LIN {X 0,Y 293.169,Z 768.015,A -85,B 0,C 180,E1 -18492.171,E2 -18492.171} C_VEL
LIN {X 0,Y 292.297,Z 765.8,A -85,B 0,C 180,E1 -18494.106,E2 -18494.106} C_VEL
LIN {X 0,Y 291.883,Z 764.889,A -85,B 0,C 180,E1 -18496.257,E2 -18496.257} C_VEL
LIN {X 0,Y 292.536,Z 764.782,A -85,B 0,C 180,E1 -18498.796,E2 -18498.796} C_VEL
LIN {X 0,Y 294.22,Z 766.186,A -85,B 0,C 180,E1 -18501.347,E2 -18501.347} C_VEL
LIN {X 0,Y 294.782,Z 766.996,A -85,B 0,C 180,E1 -18501.989,E2 -18501.989} C_VEL
LIN {X 0,Y 296.752,Z 771.019,A -85,B 0,C 180,E1 -18504.014,E2 -18504.014} C_VEL
LIN {X 0,Y 298.93,Z 775.634,A -85,B 0,C 180,E1 -18505.733,E2 -18505.733} C_VEL
LIN {X 0,Y 299.613,Z 777.365,A -85,B 0,C 180,E1 -18506.216,E2 -18506.216} C_VEL
LIN {X 0,Y 294.851,Z 808.828,A -85,B 0,C 180,E1 -18507.724,E2 -18507.724} C_VEL
LIN {X 0,Y 292.822,Z 825.485,A -85,B 0,C 180,E1 -18508.733,E2 -18508.733} C_VEL
LIN {X 0,Y 291.112,Z 835.939,A -85,B 0,C 180,E1 -18509.537,E2 -18509.537} C_VEL
LIN {X 0,Y 288.763,Z 847.798,A -85,B 0,C 180,E1 -18510.672,E2 -18510.672} C_VEL
LIN {X 0,Y 285.703,Z 859.648,A -85,B 0,C 180,E1 -18512.136,E2 -18512.136} C_VEL
LIN {X 0,Y 283.074,Z 868.365,A -85,B 0,C 180,E1 -18513.455,E2 -18513.455} C_VEL
LIN {X 0,Y 280.555,Z 875.778,A -85,B 0,C 180,E1 -18514.795,E2 -18514.795} C_VEL
LIN {X 0,Y 277.606,Z 883.425,A -85,B 0,C 180,E1 -18516.468,E2 -18516.468} C_VEL
LIN {X 0,Y 275.249,Z 888.923,A -85,B 0,C 180,E1 -18517.876,E2 -18517.876} C_VEL
LIN {X 0,Y 272.596,Z 894.53,A -85,B 0,C 180,E1 -18519.632,E2 -18519.632} C_VEL
LIN {X 0,Y 269.635,Z 899.978,A -85,B 0,C 180,E1 -18521.773,E2 -18521.773} C_VEL
LIN {X 0,Y 266.922,Z 904.27,A -85,B 0,C 180,E1 -18523.951,E2 -18523.951} C_VEL
LIN {X 0,Y 264.533,Z 907.404,A -85,B 0,C 180,E1 -18526.166,E2 -18526.166} C_VEL
LIN {X 0,Y 263.113,Z 908.967,A -85,B 0,C 180,E1 -18527.661,E2 -18527.661} C_VEL
LIN {X 0,Y 261.774,Z 910.083,A -85,B 0,C 180,E1 -18529.168,E2 -18529.168} C_VEL
LIN {X 0,Y 259.678,Z 910.938,A -85,B 0,C 180,E1 -18532.223,E2 -18532.223} C_VEL
LIN {X 0,Y 258.847,Z 910.711,A -85,B 0,C 180,E1 -18533.765,E2 -18533.765} C_VEL
LIN {X 0,Y 258.245,Z 910.062,A -85,B 0,C 180,E1 -18535.317,E2 -18535.317} C_VEL
LIN {X 0,Y 257.539,Z 908.966,A -85,B 0,C 180,E1 -18536.871,E2 -18536.871} C_VEL
LIN {X 0,Y 257.125,Z 907.432,A -85,B 0,C 180,E1 -18538.434,E2 -18538.434} C_VEL
LIN {X 0,Y 256.51,Z 904.341,A -85,B 0,C 180,E1 -18540.785,E2 -18540.785} C_VEL
LIN {X 0,Y 256.12,Z 900.192,A -85,B 0,C 180,E1 -18543.146,E2 -18543.146} C_VEL
LIN {X 0,Y 256.313,Z 893.788,A -85,B 0,C 180,E1 -18545.902,E2 -18545.902} C_VEL
LIN {X 0,Y 256.713,Z 886.811,A -85,B 0,C 180,E1 -18548.264,E2 -18548.264} C_VEL
LIN {X 0,Y 257.046,Z 880.2,A -85,B 0,C 180,E1 -18550.133,E2 -18550.133} C_VEL
LIN {X 0,Y 257.479,Z 873.243,A -85,B 0,C 180,E1 -18551.813,E2 -18551.813} C_VEL
LIN {X 0,Y 258.123,Z 864.599,A -85,B 0,C 180,E1 -18553.582,E2 -18553.582} C_VEL
LIN {X 0,Y 258.704,Z 855.499,A -85,B 0,C 180,E1 -18555.158,E2 -18555.158} C_VEL
LIN {X 0,Y 259.349,Z 846.095,A -85,B 0,C 180,E1 -18556.531,E2 -18556.531} C_VEL
LIN {X 0,Y 259.959,Z 836.514,A -85,B 0,C 180,E1 -18557.707,E2 -18557.707} C_VEL
LIN {X 0,Y 260.523,Z 826.952,A -85,B 0,C 180,E1 -18558.684,E2 -18558.684} C_VEL
LIN {X 0,Y 260.988,Z 815.785,A -85,B 0,C 180,E1 -18559.601,E2 -18559.601} C_VEL
LIN {X 0,Y 261.302,Z 804.987,A -85,B 0,C 180,E1 -18560.287,E2 -18560.287} C_VEL
LIN {X 0,Y 261.675,Z 788.222,A -85,B 0,C 180,E1 -18561.053,E2 -18561.053} C_VEL
LIN {X 0,Y 262.992,Z 743.404,A -85,B 0,C 180,E1 -18562.898,E2 -18562.898} C_VEL
LIN {X 0,Y 256.201,Z 720.571,A -85,B 0,C 180,E1 -18564.225,E2 -18564.225} C_VEL
LIN {X 0,Y 256.107,Z 720.581,A -85,B 0,C 180,E1 -18568.568,E2 -18568.568} C_VEL
LIN {X 0,Y 256.095,Z 720.583,A -85,B 0,C 180,E1 -18571.695,E2 -18571.695} C_VEL
LIN {X 0,Y 256.104,Z 720.582,A -85,B 0,C 180,E1 -18575.19,E2 -18575.19} C_VEL
LIN {X 0,Y 256.089,Z 720.581,A -85,B 0,C 180,E1 -18579.139,E2 -18579.139} C_VEL
LIN {X 0,Y 256.046,Z 720.585,A -85,B 0,C 180,E1 -18583.331,E2 -18583.331} C_VEL
LIN {X 0,Y 256.056,Z 720.583,A -85,B 0,C 180,E1 -18587.823,E2 -18587.823} C_VEL
LIN {X 0,Y 256.086,Z 720.578,A -85,B 0,C 180,E1 -18590.85,E2 -18590.85} C_VEL
LIN {X 0,Y 256.1,Z 720.577,A -85,B 0,C 180,E1 -18594.8,E2 -18594.8} C_VEL
LIN {X 0,Y 256.118,Z 720.772,A -85,B 0,C 180,E1 -18598.348,E2 -18598.348} C_VEL
LIN {X 0,Y 257.16,Z 723.493,A -85,B 0,C 180,E1 -18598.585,E2 -18598.585} C_VEL
LIN {X 0,Y 258.744,Z 726.144,A -85,B 0,C 180,E1 -18598.893,E2 -18598.893} C_VEL
LIN {X 0,Y 266.211,Z 739.942,A -85,B 0,C 180,E1 -18600.322,E2 -18600.322} C_VEL
LIN {X 0,Y 273.123,Z 754.427,A -85,B 0,C 180,E1 -18601.608,E2 -18601.608} C_VEL
LIN {X 0,Y 273.856,Z 756.115,A -85,B 0,C 180,E1 -18601.745,E2 -18601.745} C_VEL
LIN {X 0,Y 272.925,Z 794.728,A -85,B 0,C 180,E1 -18602.771,E2 -18602.771} C_VEL
LIN {X 0,Y 272.718,Z 809.458,A -85,B 0,C 180,E1 -18603.281,E2 -18603.281} C_VEL
LIN {X 0,Y 272.187,Z 821.386,A -85,B 0,C 180,E1 -18603.954,E2 -18603.954} C_VEL
LIN {X 0,Y 271.062,Z 834.416,A -85,B 0,C 180,E1 -18605.002,E2 -18605.002} C_VEL
LIN {X 0,Y 269.714,Z 845.924,A -85,B 0,C 180,E1 -18606.238,E2 -18606.238} C_VEL
LIN {X 0,Y 268.04,Z 856.353,A -85,B 0,C 180,E1 -18607.645,E2 -18607.645} C_VEL
LIN {X 0,Y 266.537,Z 865.181,A -85,B 0,C 180,E1 -18609.138,E2 -18609.138} C_VEL
LIN {X 0,Y 264.837,Z 874.215,A -85,B 0,C 180,E1 -18611.02,E2 -18611.02} C_VEL
LIN {X 0,Y 262.82,Z 882.996,A -85,B 0,C 180,E1 -18613.284,E2 -18613.284} C_VEL
LIN {X 0,Y 260.98,Z 890.664,A -85,B 0,C 180,E1 -18615.803,E2 -18615.803} C_VEL
LIN {X 0,Y 259.741,Z 896.427,A -85,B 0,C 180,E1 -18618.282,E2 -18618.282} C_VEL
LIN {X 0,Y 259.045,Z 899.362,A -85,B 0,C 180,E1 -18619.833,E2 -18619.833} C_VEL
LIN {X 0,Y 257.846,Z 902.921,A -85,B 0,C 180,E1 -18622.157,E2 -18622.157} C_VEL
LIN {X 0,Y 257.338,Z 904.743,A -85,B 0,C 180,E1 -18623.718,E2 -18623.718} C_VEL
LIN {X 0,Y 256.95,Z 907.051,A -85,B 0,C 180,E1 -18626.854,E2 -18626.854} C_VEL
LIN {X 0,Y 256.667,Z 907.89,A -85,B 0,C 180,E1 -18629.99,E2 -18629.99} C_VEL
LIN {X 0,Y 256.946,Z 907.124,A -85,B 0,C 180,E1 -18633.125,E2 -18633.125} C_VEL
LIN {X 0,Y 257.317,Z 904.893,A -85,B 0,C 180,E1 -18636.261,E2 -18636.261} C_VEL
LIN {X 0,Y 258.168,Z 902.073,A -85,B 0,C 180,E1 -18638.6,E2 -18638.6} C_VEL
LIN {X 0,Y 259.312,Z 898.243,A -85,B 0,C 180,E1 -18640.925,E2 -18640.925} C_VEL
LIN {X 0,Y 260.559,Z 892.768,A -85,B 0,C 180,E1 -18643.489,E2 -18643.489} C_VEL
LIN {X 0,Y 262.202,Z 885.953,A -85,B 0,C 180,E1 -18645.935,E2 -18645.935} C_VEL
LIN {X 0,Y 264.102,Z 877.921,A -85,B 0,C 180,E1 -18648.209,E2 -18648.209} C_VEL
LIN {X 0,Y 265.782,Z 869.698,A -85,B 0,C 180,E1 -18650.094,E2 -18650.094} C_VEL
LIN {X 0,Y 267.597,Z 859.522,A -85,B 0,C 180,E1 -18651.966,E2 -18651.966} C_VEL
LIN {X 0,Y 269.347,Z 849.047,A -85,B 0,C 180,E1 -18653.488,E2 -18653.488} C_VEL
LIN {X 0,Y 270.844,Z 837.769,A -85,B 0,C 180,E1 -18654.788,E2 -18654.788} C_VEL
LIN {X 0,Y 272.079,Z 825.822,A -85,B 0,C 180,E1 -18655.829,E2 -18655.829} C_VEL
LIN {X 0,Y 272.637,Z 813.644,A -85,B 0,C 180,E1 -18656.629,E2 -18656.629} C_VEL
LIN {X 0,Y 272.938,Z 800.891,A -85,B 0,C 180,E1 -18657.169,E2 -18657.169} C_VEL
LIN {X 0,Y 273.85,Z 760.256,A -85,B 0,C 180,E1 -18658.263,E2 -18658.263} C_VEL
LIN {X 0,Y 273.819,Z 755.874,A -85,B 0,C 180,E1 -18658.396,E2 -18658.396} C_VEL
LIN {X 0,Y 266.835,Z 741.021,A -85,B 0,C 180,E1 -18659.697,E2 -18659.697} C_VEL
LIN {X 0,Y 259.331,Z 727.24,A -85,B 0,C 180,E1 -18661.126,E2 -18661.126} C_VEL
LIN {X 0,Y 256.33,Z 721.817,A -85,B 0,C 180,E1 -18661.725,E2 -18661.725} C_VEL
LIN {X 0,Y 256.065,Z 720.589,A -85,B 0,C 180,E1 -18661.825,E2 -18661.825} C_VEL
LIN {X 0,Y 256.09,Z 720.585,A -85,B 0,C 180,E1 -18665.176,E2 -18665.176} C_VEL
LIN {X 0,Y 256.074,Z 720.569,A -85,B 0,C 180,E1 -18669.125,E2 -18669.125} C_VEL
LIN {X 0,Y 256.102,Z 720.573,A -85,B 0,C 180,E1 -18673.301,E2 -18673.301} C_VEL
LIN {X 0,Y 256.117,Z 720.579,A -85,B 0,C 180,E1 -18677.788,E2 -18677.788} C_VEL
LIN {X 0,Y 256.063,Z 720.583,A -85,B 0,C 180,E1 -18680.856,E2 -18680.856} C_VEL
LIN {X 0,Y 256.071,Z 720.583,A -85,B 0,C 180,E1 -18684.805,E2 -18684.805} C_VEL
LIN {X 0,Y 256.04,Z 720.59,A -85,B 0,C 180,E1 -18688.565,E2 -18688.565} C_VEL
LIN {X 0,Y 256.083,Z 720.578,A -85,B 0,C 180,E1 -18692.189,E2 -18692.189} C_VEL
LIN {X 0,Y 256.085,Z 720.576,A -85,B 0,C 180,E1 -18695.691,E2 -18695.691} C_VEL
LIN {X 0,Y 256.105,Z 720.583,A -85,B 0,C 180,E1 -18699.099,E2 -18699.099} C_VEL
LIN {X 0,Y 256.218,Z 720.56,A -85,B 0,C 180,E1 -18704.08,E2 -18704.08} C_VEL
LIN {X 0,Y 256.246,Z 720.551,A -85,B 0,C 180,E1 -18708.931,E2 -18708.931} C_VEL
LIN {X 0,Y 256.33,Z 720.542,A -85,B 0,C 180,E1 -18710.1,E2 -18710.1} C_VEL
LIN {X 0,Y 255.761,Z 720.627,A -85,B 0,C 180,E1 -18711.411,E2 -18711.411} C_VEL
LIN {X 0,Y 252.905,Z 720.983,A -85,B 0,C 180,E1 -18713.546,E2 -18713.546} C_VEL
LIN {X 0,Y 250.46,Z 721.279,A -85,B 0,C 180,E1 -18715.286,E2 -18715.286} C_VEL
LIN {X 0,Y 249.472,Z 721.398,A -85,B 0,C 180,E1 -18716.636,E2 -18716.636} C_VEL
LIN {X 0,Y 249.428,Z 721.404,A -85,B 0,C 180,E1 -18717.093,E2 -18717.093} C_VEL
LIN {X 0,Y 249.67,Z 721.389,A -85,B 0,C 180,E1 -18720,E2 -18720} C_VEL
LIN {X 0,Y 249.401,Z 721.408,A -85,B 0,C 180,E1 -18723.231,E2 -18723.231} C_VEL
LIN {X 0,Y 249.406,Z 721.412,A -85,B 0,C 180,E1 -18728.1,E2 -18728.1} C_VEL
LIN {X 0,Y 249.189,Z 721.445,A -85,B 0,C 180,E1 -18731.386,E2 -18731.386} C_VEL
LIN {X 0,Y 249.158,Z 721.445,A -85,B 0,C 180,E1 -18736.507,E2 -18736.507} C_VEL
LIN {X 0,Y 249.028,Z 721.452,A -85,B 0,C 180,E1 -18741.524,E2 -18741.524} C_VEL
LIN {X 0,Y 249.073,Z 721.448,A -85,B 0,C 180,E1 -18745.487,E2 -18745.487} C_VEL
LIN {X 0,Y 249.019,Z 721.464,A -85,B 0,C 180,E1 -18748.996,E2 -18748.996} C_VEL
LIN {X 0,Y 248.984,Z 721.47,A -85,B 0,C 180,E1 -18752.433,E2 -18752.433} C_VEL
LIN {X 0,Y 249.025,Z 721.464,A -85,B 0,C 180,E1 -18756.346,E2 -18756.346} C_VEL
LIN {X 0,Y 249.039,Z 721.452,A -85,B 0,C 180,E1 -18760.472,E2 -18760.472} C_VEL
LIN {X 0,Y 249.032,Z 721.47,A -85,B 0,C 180,E1 -18764.321,E2 -18764.321} C_VEL
LIN {X 0,Y 252.137,Z 732.401,A -85,B 0,C 180,E1 -18768.349,E2 -18768.349} C_VEL
LIN {X 0,Y 254.654,Z 742.514,A -85,B 0,C 180,E1 -18771.768,E2 -18771.768} C_VEL
LIN {X 0,Y 256.98,Z 753.129,A -85,B 0,C 180,E1 -18775.13,E2 -18775.13} C_VEL
LIN {X 0,Y 257.957,Z 759.353,A -85,B 0,C 180,E1 -18776.997,E2 -18776.997} C_VEL
LIN {X 0,Y 257.44,Z 762.214,A -85,B 0,C 180,E1 -18777.75,E2 -18777.75} C_VEL
LIN {X 0,Y 261.25,Z 791.203,A -85,B 0,C 180,E1 -18779.183,E2 -18779.183} C_VEL
LIN {X 0,Y 264.207,Z 821.563,A -85,B 0,C 180,E1 -18780.474,E2 -18780.474} C_VEL
LIN {X 0,Y 265.313,Z 838.589,A -85,B 0,C 180,E1 -18781.116,E2 -18781.116} C_VEL
LIN {X 0,Y 264.068,Z 874.188,A -85,B 0,C 180,E1 -18782.092,E2 -18782.092} C_VEL
LIN {X 0,Y 262.845,Z 887.976,A -85,B 0,C 180,E1 -18782.755,E2 -18782.755} C_VEL
LIN {X 0,Y 261.319,Z 900.557,A -85,B 0,C 180,E1 -18783.67,E2 -18783.67} C_VEL
LIN {X 0,Y 259.44,Z 911.71,A -85,B 0,C 180,E1 -18784.758,E2 -18784.758} C_VEL
LIN {X 0,Y 257.126,Z 923.35,A -85,B 0,C 180,E1 -18786.237,E2 -18786.237} C_VEL
LIN {X 0,Y 254.911,Z 933.879,A -85,B 0,C 180,E1 -18787.949,E2 -18787.949} C_VEL
LIN {X 0,Y 252.942,Z 942.516,A -85,B 0,C 180,E1 -18789.69,E2 -18789.69} C_VEL
LIN {X 0,Y 251.298,Z 950.546,A -85,B 0,C 180,E1 -18791.674,E2 -18791.674} C_VEL
LIN {X 0,Y 249.89,Z 957.229,A -85,B 0,C 180,E1 -18793.678,E2 -18793.678} C_VEL
LIN {X 0,Y 248.763,Z 963.864,A -85,B 0,C 180,E1 -18796.117,E2 -18796.117} C_VEL
LIN {X 0,Y 248.083,Z 969.178,A -85,B 0,C 180,E1 -18798.574,E2 -18798.574} C_VEL
LIN {X 0,Y 247.895,Z 973.364,A -85,B 0,C 180,E1 -18801.041,E2 -18801.041} C_VEL
LIN {X 0,Y 248.045,Z 976.5,A -85,B 0,C 180,E1 -18803.504,E2 -18803.504} C_VEL
LIN {X 0,Y 248.285,Z 978.015,A -85,B 0,C 180,E1 -18805.14,E2 -18805.14} C_VEL
LIN {X 0,Y 248.498,Z 979.1,A -85,B 0,C 180,E1 -18806.768,E2 -18806.768} C_VEL
LIN {X 0,Y 248.69,Z 979.769,A -85,B 0,C 180,E1 -18808.391,E2 -18808.391} C_VEL
LIN {X 0,Y 248.88,Z 980.017,A -85,B 0,C 180,E1 -18810.011,E2 -18810.011} C_VEL
LIN {X 0,Y 248.689,Z 979.752,A -85,B 0,C 180,E1 -18811.63,E2 -18811.63} C_VEL
LIN {X 0,Y 248.494,Z 979.072,A -85,B 0,C 180,E1 -18813.253,E2 -18813.253} C_VEL
LIN {X 0,Y 248.273,Z 977.974,A -85,B 0,C 180,E1 -18814.882,E2 -18814.882} C_VEL
LIN {X 0,Y 247.98,Z 975.552,A -85,B 0,C 180,E1 -18817.281,E2 -18817.281} C_VEL
LIN {X 0,Y 248.209,Z 969.865,A -85,B 0,C 180,E1 -18822.271,E2 -18822.271} C_VEL
LIN {X 0,Y 249.089,Z 966.281,A -85,B 0,C 180,E1 -18824.72,E2 -18824.72} C_VEL
LIN {X 0,Y 250.863,Z 960.397,A -85,B 0,C 180,E1 -18827.727,E2 -18827.727} C_VEL
LIN {X 0,Y 253.032,Z 955.019,A -85,B 0,C 180,E1 -18829.902,E2 -18829.902} C_VEL
LIN {X 0,Y 255.726,Z 948.036,A -85,B 0,C 180,E1 -18832.212,E2 -18832.212} C_VEL
LIN {X 0,Y 258.534,Z 941.236,A -85,B 0,C 180,E1 -18834.074,E2 -18834.074} C_VEL
LIN {X 0,Y 262.541,Z 931.503,A -85,B 0,C 180,E1 -18836.221,E2 -18836.221} C_VEL
LIN {X 0,Y 265.938,Z 922.997,A -85,B 0,C 180,E1 -18837.77,E2 -18837.77} C_VEL
LIN {X 0,Y 269.691,Z 912.988,A -85,B 0,C 180,E1 -18839.259,E2 -18839.259} C_VEL
LIN {X 0,Y 273.427,Z 902.615,A -85,B 0,C 180,E1 -18840.516,E2 -18840.516} C_VEL
LIN {X 0,Y 276.85,Z 891.854,A -85,B 0,C 180,E1 -18841.581,E2 -18841.581} C_VEL
LIN {X 0,Y 279.987,Z 880.8,A -85,B 0,C 180,E1 -18842.457,E2 -18842.457} C_VEL
LIN {X 0,Y 283.535,Z 866.175,A -85,B 0,C 180,E1 -18843.373,E2 -18843.373} C_VEL
LIN {X 0,Y 287.026,Z 844.8,A -85,B 0,C 180,E1 -18844.388,E2 -18844.388} C_VEL
LIN {X 0,Y 289.011,Z 825.027,A -85,B 0,C 180,E1 -18845.714,E2 -18845.714} C_VEL
LIN {X 0,Y 290.09,Z 809.979,A -85,B 0,C 180,E1 -18847.027,E2 -18847.027} C_VEL
LIN {X 0,Y 291.339,Z 791.88,A -85,B 0,C 180,E1 -18848.883,E2 -18848.883} C_VEL
LIN {X 0,Y 291.656,Z 785.798,A -85,B 0,C 180,E1 -18849.649,E2 -18849.649} C_VEL
LIN {X 0,Y 291.112,Z 776.146,A -85,B 0,C 180,E1 -18852.13,E2 -18852.13} C_VEL
LIN {X 0,Y 291.05,Z 774.422,A -85,B 0,C 180,E1 -18852.673,E2 -18852.673} C_VEL
LIN {X 0,Y 290.487,Z 772.629,A -85,B 0,C 180,E1 -18854.213,E2 -18854.213} C_VEL
LIN {X 0,Y 290.166,Z 771.711,A -85,B 0,C 180,E1 -18856.613,E2 -18856.613} C_VEL
LIN {X 0,Y 290.991,Z 771.836,A -85,B 0,C 180,E1 -18859.3,E2 -18859.3} C_VEL
LIN {X 0,Y 292.489,Z 773.149,A -85,B 0,C 180,E1 -18861.409,E2 -18861.409} C_VEL
LIN {X 0,Y 294.44,Z 777.474,A -85,B 0,C 180,E1 -18863.641,E2 -18863.641} C_VEL
LIN {X 0,Y 296.109,Z 781.305,A -85,B 0,C 180,E1 -18865.099,E2 -18865.099} C_VEL
LIN {X 0,Y 291.176,Z 812.172,A -85,B 0,C 180,E1 -18866.642,E2 -18866.642} C_VEL
LIN {X 0,Y 288.986,Z 828.026,A -85,B 0,C 180,E1 -18867.654,E2 -18867.654} C_VEL
LIN {X 0,Y 286.813,Z 840.119,A -85,B 0,C 180,E1 -18868.62,E2 -18868.62} C_VEL
LIN {X 0,Y 283.873,Z 852.515,A -85,B 0,C 180,E1 -18869.911,E2 -18869.911} C_VEL
LIN {X 0,Y 281.006,Z 862.498,A -85,B 0,C 180,E1 -18871.22,E2 -18871.22} C_VEL
LIN {X 0,Y 278.195,Z 870.951,A -85,B 0,C 180,E1 -18872.545,E2 -18872.545} C_VEL
LIN {X 0,Y 275.496,Z 878.087,A -85,B 0,C 180,E1 -18873.893,E2 -18873.893} C_VEL
LIN {X 0,Y 273.201,Z 883.79,A -85,B 0,C 180,E1 -18875.14,E2 -18875.14} C_VEL
LIN {X 0,Y 270.45,Z 889.739,A -85,B 0,C 180,E1 -18876.653,E2 -18876.653} C_VEL
LIN {X 0,Y 267.54,Z 895.423,A -85,B 0,C 180,E1 -18878.422,E2 -18878.422} C_VEL
LIN {X 0,Y 264.326,Z 900.969,A -85,B 0,C 180,E1 -18880.588,E2 -18880.588} C_VEL
LIN {X 0,Y 261.376,Z 905.28,A -85,B 0,C 180,E1 -18882.796,E2 -18882.796} C_VEL
LIN {X 0,Y 259.59,Z 907.646,A -85,B 0,C 180,E1 -18884.292,E2 -18884.292} C_VEL
LIN {X 0,Y 257.943,Z 909.391,A -85,B 0,C 180,E1 -18885.805,E2 -18885.805} C_VEL
LIN {X 0,Y 255.022,Z 911.73,A -85,B 0,C 180,E1 -18888.877,E2 -18888.877} C_VEL
LIN {X 0,Y 252.781,Z 912.262,A -85,B 0,C 180,E1 -18892.009,E2 -18892.009} C_VEL
LIN {X 0,Y 251.897,Z 911.904,A -85,B 0,C 180,E1 -18893.592,E2 -18893.592} C_VEL
LIN {X 0,Y 251.266,Z 911.066,A -85,B 0,C 180,E1 -18895.187,E2 -18895.187} C_VEL
LIN {X 0,Y 250.07,Z 908.213,A -85,B 0,C 180,E1 -18898.39,E2 -18898.39} C_VEL
LIN {X 0,Y 249.444,Z 904.875,A -85,B 0,C 180,E1 -18900.807,E2 -18900.807} C_VEL
LIN {X 0,Y 249.05,Z 900.432,A -85,B 0,C 180,E1 -18903.236,E2 -18903.236} C_VEL
LIN {X 0,Y 249.168,Z 894.774,A -85,B 0,C 180,E1 -18905.666,E2 -18905.666} C_VEL
LIN {X 0,Y 249.547,Z 888.382,A -85,B 0,C 180,E1 -18907.907,E2 -18907.907} C_VEL
LIN {X 0,Y 249.854,Z 882.301,A -85,B 0,C 180,E1 -18909.716,E2 -18909.716} C_VEL
LIN {X 0,Y 250.361,Z 874.143,A -85,B 0,C 180,E1 -18911.743,E2 -18911.743} C_VEL
LIN {X 0,Y 251.016,Z 865.436,A -85,B 0,C 180,E1 -18913.561,E2 -18913.561} C_VEL
LIN {X 0,Y 251.632,Z 856.273,A -85,B 0,C 180,E1 -18915.179,E2 -18915.179} C_VEL
LIN {X 0,Y 252.255,Z 846.781,A -85,B 0,C 180,E1 -18916.593,E2 -18916.593} C_VEL
LIN {X 0,Y 252.875,Z 837.104,A -85,B 0,C 180,E1 -18917.801,E2 -18917.801} C_VEL
LIN {X 0,Y 253.496,Z 826.357,A -85,B 0,C 180,E1 -18918.907,E2 -18918.907} C_VEL
LIN {X 0,Y 253.981,Z 814.935,A -85,B 0,C 180,E1 -18919.845,E2 -18919.845} C_VEL
LIN {X 0,Y 254.342,Z 801.66,A -85,B 0,C 180,E1 -18920.667,E2 -18920.667} C_VEL
LIN {X 0,Y 255.9,Z 750.146,A -85,B 0,C 180,E1 -18922.906,E2 -18922.906} C_VEL
LIN {X 0,Y 255.927,Z 744.55,A -85,B 0,C 180,E1 -18923.151,E2 -18923.151} C_VEL
LIN {X 0,Y 249.155,Z 721.448,A -85,B 0,C 180,E1 -18924.511,E2 -18924.511} C_VEL
LIN {X 0,Y 249.054,Z 721.463,A -85,B 0,C 180,E1 -18928.966,E2 -18928.966} C_VEL
LIN {X 0,Y 249.052,Z 721.462,A -85,B 0,C 180,E1 -18932.423,E2 -18932.423} C_VEL
LIN {X 0,Y 249.037,Z 721.46,A -85,B 0,C 180,E1 -18936.345,E2 -18936.345} C_VEL
LIN {X 0,Y 249.004,Z 721.465,A -85,B 0,C 180,E1 -18940.479,E2 -18940.479} C_VEL
LIN {X 0,Y 248.986,Z 721.464,A -85,B 0,C 180,E1 -18944.884,E2 -18944.884} C_VEL
LIN {X 0,Y 249.002,Z 721.463,A -85,B 0,C 180,E1 -18947.349,E2 -18947.349} C_VEL
LIN {X 0,Y 249.066,Z 721.453,A -85,B 0,C 180,E1 -18952.194,E2 -18952.194} C_VEL
LIN {X 0,Y 249.06,Z 721.454,A -85,B 0,C 180,E1 -18956.606,E2 -18956.606} C_VEL
LIN {X 0,Y 249.029,Z 721.457,A -85,B 0,C 180,E1 -18957.292,E2 -18957.292} C_VEL
LIN {X 0,Y 250.041,Z 724.295,A -85,B 0,C 180,E1 -18957.569,E2 -18957.569} C_VEL
LIN {X 0,Y 251.872,Z 727.362,A -85,B 0,C 180,E1 -18957.946,E2 -18957.946} C_VEL
LIN {X 0,Y 258.693,Z 739.507,A -85,B 0,C 180,E1 -18959.314,E2 -18959.314} C_VEL
LIN {X 0,Y 266.732,Z 756.106,A -85,B 0,C 180,E1 -18960.882,E2 -18960.882} C_VEL
LIN {X 0,Y 267.626,Z 758.075,A -85,B 0,C 180,E1 -18961.053,E2 -18961.053} C_VEL
LIN {X 0,Y 266.696,Z 795.311,A -85,B 0,C 180,E1 -18962.067,E2 -18962.067} C_VEL
LIN {X 0,Y 266.436,Z 810.923,A -85,B 0,C 180,E1 -18962.62,E2 -18962.62} C_VEL
LIN {X 0,Y 265.806,Z 823.711,A -85,B 0,C 180,E1 -18963.386,E2 -18963.386} C_VEL
LIN {X 0,Y 264.592,Z 836.502,A -85,B 0,C 180,E1 -18964.462,E2 -18964.462} C_VEL
LIN {X 0,Y 263.111,Z 848.07,A -85,B 0,C 180,E1 -18965.757,E2 -18965.757} C_VEL
LIN {X 0,Y 261.392,Z 858.529,A -85,B 0,C 180,E1 -18967.254,E2 -18967.254} C_VEL
LIN {X 0,Y 259.577,Z 868.12,A -85,B 0,C 180,E1 -18968.968,E2 -18968.968} C_VEL
LIN {X 0,Y 257.855,Z 876.811,A -85,B 0,C 180,E1 -18970.9,E2 -18970.9} C_VEL
LIN {X 0,Y 255.798,Z 885.31,A -85,B 0,C 180,E1 -18973.223,E2 -18973.223} C_VEL
LIN {X 0,Y 254.041,Z 892.069,A -85,B 0,C 180,E1 -18975.573,E2 -18975.573} C_VEL
LIN {X 0,Y 252.863,Z 897.431,A -85,B 0,C 180,E1 -18977.958,E2 -18977.958} C_VEL
LIN {X 0,Y 252.131,Z 900.366,A -85,B 0,C 180,E1 -18979.551,E2 -18979.551} C_VEL
LIN {X 0,Y 250.886,Z 903.924,A -85,B 0,C 180,E1 -18981.938,E2 -18981.938} C_VEL
LIN {X 0,Y 250.353,Z 905.746,A -85,B 0,C 180,E1 -18983.542,E2 -18983.542} C_VEL
LIN {X 0,Y 249.934,Z 908.054,A -85,B 0,C 180,E1 -18986.766,E2 -18986.766} C_VEL
LIN {X 0,Y 249.639,Z 908.893,A -85,B 0,C 180,E1 -18989.989,E2 -18989.989} C_VEL
LIN {X 0,Y 249.929,Z 908.126,A -85,B 0,C 180,E1 -18993.213,E2 -18993.213} C_VEL
LIN {X 0,Y 250.331,Z 905.895,A -85,B 0,C 180,E1 -18996.437,E2 -18996.437} C_VEL
LIN {X 0,Y 251.222,Z 903.074,A -85,B 0,C 180,E1 -18998.84,E2 -18998.84} C_VEL
LIN {X 0,Y 252.415,Z 899.245,A -85,B 0,C 180,E1 -19001.227,E2 -19001.227} C_VEL
LIN {X 0,Y 253.73,Z 893.769,A -85,B 0,C 180,E1 -19003.859,E2 -19003.859} C_VEL
LIN {X 0,Y 255.451,Z 886.953,A -85,B 0,C 180,E1 -19006.367,E2 -19006.367} C_VEL
LIN {X 0,Y 257.435,Z 878.921,A -85,B 0,C 180,E1 -19008.698,E2 -19008.698} C_VEL
LIN {X 0,Y 259.193,Z 870.698,A -85,B 0,C 180,E1 -19010.627,E2 -19010.627} C_VEL
LIN {X 0,Y 261.092,Z 860.521,A -85,B 0,C 180,E1 -19012.543,E2 -19012.543} C_VEL
LIN {X 0,Y 262.916,Z 850.044,A -85,B 0,C 180,E1 -19014.099,E2 -19014.099} C_VEL
LIN {X 0,Y 264.481,Z 838.765,A -85,B 0,C 180,E1 -19015.427,E2 -19015.427} C_VEL
LIN {X 0,Y 265.77,Z 826.816,A -85,B 0,C 180,E1 -19016.489,E2 -19016.489} C_VEL
LIN {X 0,Y 266.379,Z 814.229,A -85,B 0,C 180,E1 -19017.33,E2 -19017.33} C_VEL
LIN {X 0,Y 266.701,Z 801.485,A -85,B 0,C 180,E1 -19017.873,E2 -19017.873} C_VEL
LIN {X 0,Y 267.6,Z 761.77,A -85,B 0,C 180,E1 -19018.969,E2 -19018.969} C_VEL
LIN {X 0,Y 267.635,Z 758.009,A -85,B 0,C 180,E1 -19019.079,E2 -19019.079} C_VEL
LIN {X 0,Y 260.781,Z 743.445,A -85,B 0,C 180,E1 -19020.413,E2 -19020.413} C_VEL
LIN {X 0,Y 252.565,Z 728.492,A -85,B 0,C 180,E1 -19022.053,E2 -19022.053} C_VEL
LIN {X 0,Y 249.317,Z 722.816,A -85,B 0,C 180,E1 -19022.732,E2 -19022.732} C_VEL
LIN {X 0,Y 249.023,Z 721.466,A -85,B 0,C 180,E1 -19022.843,E2 -19022.843} C_VEL
LIN {X 0,Y 249.042,Z 721.462,A -85,B 0,C 180,E1 -19026.327,E2 -19026.327} C_VEL
LIN {X 0,Y 249.047,Z 721.461,A -85,B 0,C 180,E1 -19030.452,E2 -19030.452} C_VEL
LIN {X 0,Y 249.055,Z 721.457,A -85,B 0,C 180,E1 -19032.803,E2 -19032.803} C_VEL
LIN {X 0,Y 249.055,Z 721.455,A -85,B 0,C 180,E1 -19037.371,E2 -19037.371} C_VEL
LIN {X 0,Y 249.006,Z 721.461,A -85,B 0,C 180,E1 -19041.615,E2 -19041.615} C_VEL
LIN {X 0,Y 249.011,Z 721.457,A -85,B 0,C 180,E1 -19045.634,E2 -19045.634} C_VEL
LIN {X 0,Y 248.995,Z 721.466,A -85,B 0,C 180,E1 -19049.465,E2 -19049.465} C_VEL
LIN {X 0,Y 249.013,Z 721.465,A -85,B 0,C 180,E1 -19053.155,E2 -19053.155} C_VEL
LIN {X 0,Y 249.004,Z 721.455,A -85,B 0,C 180,E1 -19056.725,E2 -19056.725} C_VEL
LIN {X 0,Y 249.05,Z 721.461,A -85,B 0,C 180,E1 -19060.206,E2 -19060.206} C_VEL
LIN {X 0,Y 249.144,Z 721.439,A -85,B 0,C 180,E1 -19063.615,E2 -19063.615} C_VEL
LIN {X 0,Y 249.189,Z 721.432,A -85,B 0,C 180,E1 -19068.613,E2 -19068.613} C_VEL
LIN {X 0,Y 249.406,Z 721.419,A -85,B 0,C 180,E1 -19071.9,E2 -19071.9} C_VEL
LIN {X 0,Y 249.4,Z 721.407,A -85,B 0,C 180,E1 -19076.769,E2 -19076.769} C_VEL
LIN {X 0,Y 249.428,Z 721.404,A -85,B 0,C 180,E1 -19077.093,E2 -19077.093} C_VEL
LIN {X 0,Y 249.185,Z 721.445,A -85,B 0,C 180,E1 -19077.996,E2 -19077.996} C_VEL
LIN {X 0,Y 247.887,Z 721.613,A -85,B 0,C 180,E1 -19079.33,E2 -19079.33} C_VEL
LIN {X 0,Y 243.479,Z 722.149,A -85,B 0,C 180,E1 -19082.437,E2 -19082.437} C_VEL
LIN {X 0,Y 242.348,Z 722.29,A -85,B 0,C 180,E1 -19083.829,E2 -19083.829} C_VEL
LIN {X 0,Y 242.233,Z 722.304,A -85,B 0,C 180,E1 -19084.302,E2 -19084.302} C_VEL
LIN {X 0,Y 242.365,Z 722.299,A -85,B 0,C 180,E1 -19086.661,E2 -19086.661} C_VEL
LIN {X 0,Y 242.251,Z 722.299,A -85,B 0,C 180,E1 -19090.024,E2 -19090.024} C_VEL
LIN {X 0,Y 242.089,Z 722.331,A -85,B 0,C 180,E1 -19095.146,E2 -19095.146} C_VEL
LIN {X 0,Y 242.008,Z 722.338,A -85,B 0,C 180,E1 -19098.629,E2 -19098.629} C_VEL
LIN {X 0,Y 241.954,Z 722.338,A -85,B 0,C 180,E1 -19102.186,E2 -19102.186} C_VEL
LIN {X 0,Y 242.012,Z 722.326,A -85,B 0,C 180,E1 -19105.844,E2 -19105.844} C_VEL
LIN {X 0,Y 241.954,Z 722.338,A -85,B 0,C 180,E1 -19109.59,E2 -19109.59} C_VEL
LIN {X 0,Y 241.941,Z 722.342,A -85,B 0,C 180,E1 -19113.499,E2 -19113.499} C_VEL
LIN {X 0,Y 241.964,Z 722.328,A -85,B 0,C 180,E1 -19117.587,E2 -19117.587} C_VEL
LIN {X 0,Y 241.993,Z 722.341,A -85,B 0,C 180,E1 -19121.911,E2 -19121.911} C_VEL
LIN {X 0,Y 242.012,Z 722.453,A -85,B 0,C 180,E1 -19123.384,E2 -19123.384} C_VEL
LIN {X 0,Y 244.753,Z 731.983,A -85,B 0,C 180,E1 -19127.072,E2 -19127.072} C_VEL
LIN {X 0,Y 247.302,Z 741.877,A -85,B 0,C 180,E1 -19130.608,E2 -19130.608} C_VEL
LIN {X 0,Y 249.821,Z 753.176,A -85,B 0,C 180,E1 -19134.351,E2 -19134.351} C_VEL
LIN {X 0,Y 251.089,Z 760.866,A -85,B 0,C 180,E1 -19136.745,E2 -19136.745} C_VEL
LIN {X 0,Y 251.089,Z 761.843,A -85,B 0,C 180,E1 -19136.878,E2 -19136.878} C_VEL
LIN {X 0,Y 254.901,Z 790.167,A -85,B 0,C 180,E1 -19138.328,E2 -19138.328} C_VEL
LIN {X 0,Y 258.041,Z 822.973,A -85,B 0,C 180,E1 -19139.771,E2 -19139.771} C_VEL
LIN {X 0,Y 259.076,Z 838.701,A -85,B 0,C 180,E1 -19140.387,E2 -19140.387} C_VEL
LIN {X 0,Y 257.822,Z 873.175,A -85,B 0,C 180,E1 -19141.354,E2 -19141.354} C_VEL
LIN {X 0,Y 256.558,Z 887.106,A -85,B 0,C 180,E1 -19142.039,E2 -19142.039} C_VEL
LIN {X 0,Y 254.987,Z 899.552,A -85,B 0,C 180,E1 -19142.963,E2 -19142.963} C_VEL
LIN {X 0,Y 252.716,Z 912.293,A -85,B 0,C 180,E1 -19144.258,E2 -19144.258} C_VEL
LIN {X 0,Y 250.344,Z 923.641,A -85,B 0,C 180,E1 -19145.773,E2 -19145.773} C_VEL
LIN {X 0,Y 248.073,Z 933.916,A -85,B 0,C 180,E1 -19147.527,E2 -19147.527} C_VEL
LIN {X 0,Y 245.841,Z 943.2,A -85,B 0,C 180,E1 -19149.514,E2 -19149.514} C_VEL
LIN {X 0,Y 243.801,Z 952.586,A -85,B 0,C 180,E1 -19152.043,E2 -19152.043} C_VEL
LIN {X 0,Y 242.351,Z 959.707,A -85,B 0,C 180,E1 -19154.453,E2 -19154.453} C_VEL
LIN {X 0,Y 241.257,Z 966.496,A -85,B 0,C 180,E1 -19157.392,E2 -19157.392} C_VEL
LIN {X 0,Y 240.858,Z 971.047,A -85,B 0,C 180,E1 -19159.929,E2 -19159.929} C_VEL
LIN {X 0,Y 240.945,Z 974.715,A -85,B 0,C 180,E1 -19162.627,E2 -19162.627} C_VEL
LIN {X 0,Y 241.219,Z 977.003,A -85,B 0,C 180,E1 -19164.997,E2 -19164.997} C_VEL
LIN {X 0,Y 241.441,Z 978.092,A -85,B 0,C 180,E1 -19166.674,E2 -19166.674} C_VEL
LIN {X 0,Y 241.641,Z 978.763,A -85,B 0,C 180,E1 -19168.345,E2 -19168.345} C_VEL
LIN {X 0,Y 241.845,Z 979.013,A -85,B 0,C 180,E1 -19170.011,E2 -19170.011} C_VEL
LIN {X 0,Y 241.639,Z 978.746,A -85,B 0,C 180,E1 -19171.678,E2 -19171.678} C_VEL
LIN {X 0,Y 241.437,Z 978.063,A -85,B 0,C 180,E1 -19173.348,E2 -19173.348} C_VEL
LIN {X 0,Y 241.207,Z 976.961,A -85,B 0,C 180,E1 -19175.025,E2 -19175.025} C_VEL
LIN {X 0,Y 240.913,Z 974.741,A -85,B 0,C 180,E1 -19177.314,E2 -19177.314} C_VEL
LIN {X 0,Y 241.476,Z 968.079,A -85,B 0,C 180,E1 -19183.474,E2 -19183.474} C_VEL
LIN {X 0,Y 242.58,Z 964.425,A -85,B 0,C 180,E1 -19185.986,E2 -19185.986} C_VEL
LIN {X 0,Y 244.305,Z 959.8,A -85,B 0,C 180,E1 -19188.458,E2 -19188.458} C_VEL
LIN {X 0,Y 247.202,Z 953.051,A -85,B 0,C 180,E1 -19191.263,E2 -19191.263} C_VEL
LIN {X 0,Y 250.358,Z 945.994,A -85,B 0,C 180,E1 -19193.59,E2 -19193.59} C_VEL
LIN {X 0,Y 253.433,Z 939.201,A -85,B 0,C 180,E1 -19195.467,E2 -19195.467} C_VEL
LIN {X 0,Y 257.036,Z 931.24,A -85,B 0,C 180,E1 -19197.267,E2 -19197.267} C_VEL
LIN {X 0,Y 261.464,Z 920.953,A -85,B 0,C 180,E1 -19199.166,E2 -19199.166} C_VEL
LIN {X 0,Y 265.515,Z 910.995,A -85,B 0,C 180,E1 -19200.642,E2 -19200.642} C_VEL
LIN {X 0,Y 269.983,Z 899.2,A -85,B 0,C 180,E1 -19202.041,E2 -19202.041} C_VEL
LIN {X 0,Y 274.195,Z 886.639,A -85,B 0,C 180,E1 -19203.23,E2 -19203.23} C_VEL
LIN {X 0,Y 278.474,Z 871.524,A -85,B 0,C 180,E1 -19204.28,E2 -19204.28} C_VEL
LIN {X 0,Y 281.388,Z 858.316,A -85,B 0,C 180,E1 -19205.015,E2 -19205.015} C_VEL
LIN {X 0,Y 283.791,Z 843.789,A -85,B 0,C 180,E1 -19205.733,E2 -19205.733} C_VEL
LIN {X 0,Y 285.843,Z 825.691,A -85,B 0,C 180,E1 -19207.01,E2 -19207.01} C_VEL
LIN {X 0,Y 287.083,Z 811.963,A -85,B 0,C 180,E1 -19208.256,E2 -19208.256} C_VEL
LIN {X 0,Y 288.64,Z 795.617,A -85,B 0,C 180,E1 -19209.955,E2 -19209.955} C_VEL
LIN {X 0,Y 289.119,Z 790.284,A -85,B 0,C 180,E1 -19210.64,E2 -19210.64} C_VEL
LIN {X 0,Y 289.012,Z 781.145,A -85,B 0,C 180,E1 -19213.048,E2 -19213.048} C_VEL
LIN {X 0,Y 288.697,Z 779.529,A -85,B 0,C 180,E1 -19214.256,E2 -19214.256} C_VEL
LIN {X 0,Y 288.381,Z 778.657,A -85,B 0,C 180,E1 -19216.117,E2 -19216.117} C_VEL
LIN {X 0,Y 289.185,Z 778.688,A -85,B 0,C 180,E1 -19219.226,E2 -19219.226} C_VEL
LIN {X 0,Y 290.41,Z 779.796,A -85,B 0,C 180,E1 -19221.112,E2 -19221.112} C_VEL
LIN {X 0,Y 292.078,Z 783.842,A -85,B 0,C 180,E1 -19223.217,E2 -19223.217} C_VEL
LIN {X 0,Y 292.863,Z 785.755,A -85,B 0,C 180,E1 -19224.016,E2 -19224.016} C_VEL
LIN {X 0,Y 288.01,Z 813.907,A -85,B 0,C 180,E1 -19225.434,E2 -19225.434} C_VEL
LIN {X 0,Y 285.538,Z 829.966,A -85,B 0,C 180,E1 -19226.478,E2 -19226.478} C_VEL
LIN {X 0,Y 283.395,Z 840.885,A -85,B 0,C 180,E1 -19227.359,E2 -19227.359} C_VEL
LIN {X 0,Y 280.271,Z 853.308,A -85,B 0,C 180,E1 -19228.646,E2 -19228.646} C_VEL
LIN {X 0,Y 277.014,Z 863.861,A -85,B 0,C 180,E1 -19230.024,E2 -19230.024} C_VEL
LIN {X 0,Y 273.971,Z 872.257,A -85,B 0,C 180,E1 -19231.355,E2 -19231.355} C_VEL
LIN {X 0,Y 270.753,Z 880.201,A -85,B 0,C 180,E1 -19232.873,E2 -19232.873} C_VEL
LIN {X 0,Y 267.847,Z 886.609,A -85,B 0,C 180,E1 -19234.346,E2 -19234.346} C_VEL
LIN {X 0,Y 264.528,Z 893.02,A -85,B 0,C 180,E1 -19236.099,E2 -19236.099} C_VEL
LIN {X 0,Y 261.475,Z 898.368,A -85,B 0,C 180,E1 -19237.896,E2 -19237.896} C_VEL
LIN {X 0,Y 258.055,Z 903.553,A -85,B 0,C 180,E1 -19240.097,E2 -19240.097} C_VEL
LIN {X 0,Y 254.962,Z 907.61,A -85,B 0,C 180,E1 -19242.349,E2 -19242.349} C_VEL
LIN {X 0,Y 253.069,Z 909.705,A -85,B 0,C 180,E1 -19243.876,E2 -19243.876} C_VEL
LIN {X 0,Y 251.349,Z 911.374,A -85,B 0,C 180,E1 -19245.425,E2 -19245.425} C_VEL
LIN {X 0,Y 248.237,Z 913.276,A -85,B 0,C 180,E1 -19248.569,E2 -19248.569} C_VEL
LIN {X 0,Y 246.936,Z 913.666,A -85,B 0,C 180,E1 -19250.168,E2 -19250.168} C_VEL
LIN {X 0,Y 245.881,Z 913.549,A -85,B 0,C 180,E1 -19251.784,E2 -19251.784} C_VEL
LIN {X 0,Y 244.946,Z 913.002,A -85,B 0,C 180,E1 -19253.41,E2 -19253.41} C_VEL
LIN {X 0,Y 244.285,Z 912.04,A -85,B 0,C 180,E1 -19255.049,E2 -19255.049} C_VEL
LIN {X 0,Y 243.008,Z 908.811,A -85,B 0,C 180,E1 -19258.343,E2 -19258.343} C_VEL
LIN {X 0,Y 242.353,Z 905.237,A -85,B 0,C 180,E1 -19260.831,E2 -19260.831} C_VEL
LIN {X 0,Y 241.979,Z 900.557,A -85,B 0,C 180,E1 -19263.33,E2 -19263.33} C_VEL
LIN {X 0,Y 242.052,Z 895.741,A -85,B 0,C 180,E1 -19265.415,E2 -19265.415} C_VEL
LIN {X 0,Y 242.373,Z 889.973,A -85,B 0,C 180,E1 -19267.498,E2 -19267.498} C_VEL
LIN {X 0,Y 242.734,Z 883.105,A -85,B 0,C 180,E1 -19269.583,E2 -19269.583} C_VEL
LIN {X 0,Y 243.25,Z 874.92,A -85,B 0,C 180,E1 -19271.668,E2 -19271.668} C_VEL
LIN {X 0,Y 243.864,Z 866.187,A -85,B 0,C 180,E1 -19273.542,E2 -19273.542} C_VEL
LIN {X 0,Y 244.536,Z 857.02,A -85,B 0,C 180,E1 -19275.204,E2 -19275.204} C_VEL
LIN {X 0,Y 245.132,Z 847.44,A -85,B 0,C 180,E1 -19276.661,E2 -19276.661} C_VEL
LIN {X 0,Y 245.812,Z 837.696,A -85,B 0,C 180,E1 -19277.9,E2 -19277.9} C_VEL
LIN {X 0,Y 246.439,Z 826.843,A -85,B 0,C 180,E1 -19279.037,E2 -19279.037} C_VEL
LIN {X 0,Y 246.894,Z 815.669,A -85,B 0,C 180,E1 -19279.974,E2 -19279.974} C_VEL
LIN {X 0,Y 247.293,Z 801.508,A -85,B 0,C 180,E1 -19280.862,E2 -19280.862} C_VEL
LIN {X 0,Y 248.928,Z 749.939,A -85,B 0,C 180,E1 -19283.175,E2 -19283.175} C_VEL
LIN {X 0,Y 248.971,Z 745.863,A -85,B 0,C 180,E1 -19283.36,E2 -19283.36} C_VEL
LIN {X 0,Y 242.092,Z 722.327,A -85,B 0,C 180,E1 -19284.792,E2 -19284.792} C_VEL
LIN {X 0,Y 241.991,Z 722.341,A -85,B 0,C 180,E1 -19289.586,E2 -19289.586} C_VEL
LIN {X 0,Y 242.005,Z 722.336,A -85,B 0,C 180,E1 -19293.489,E2 -19293.489} C_VEL
LIN {X 0,Y 242.009,Z 722.337,A -85,B 0,C 180,E1 -19297.579,E2 -19297.579} C_VEL
LIN {X 0,Y 241.932,Z 722.342,A -85,B 0,C 180,E1 -19301.924,E2 -19301.924} C_VEL
LIN {X 0,Y 241.924,Z 722.342,A -85,B 0,C 180,E1 -19306.574,E2 -19306.574} C_VEL
LIN {X 0,Y 242.016,Z 722.331,A -85,B 0,C 180,E1 -19311.635,E2 -19311.635} C_VEL
LIN {X 0,Y 242.032,Z 722.344,A -85,B 0,C 180,E1 -19316.238,E2 -19316.238} C_VEL
LIN {X 0,Y 243.019,Z 725.147,A -85,B 0,C 180,E1 -19316.498,E2 -19316.498} C_VEL
LIN {X 0,Y 244.7,Z 727.954,A -85,B 0,C 180,E1 -19316.866,E2 -19316.866} C_VEL
LIN {X 0,Y 251.456,Z 739.769,A -85,B 0,C 180,E1 -19318.298,E2 -19318.298} C_VEL
LIN {X 0,Y 259.573,Z 755.848,A -85,B 0,C 180,E1 -19319.952,E2 -19319.952} C_VEL
LIN {X 0,Y 261.429,Z 760.084,A -85,B 0,C 180,E1 -19320.33,E2 -19320.33} C_VEL
LIN {X 0,Y 260.492,Z 795.658,A -85,B 0,C 180,E1 -19321.32,E2 -19321.32} C_VEL
LIN {X 0,Y 260.222,Z 811.645,A -85,B 0,C 180,E1 -19321.895,E2 -19321.895} C_VEL
LIN {X 0,Y 259.537,Z 824.723,A -85,B 0,C 180,E1 -19322.691,E2 -19322.691} C_VEL
LIN {X 0,Y 258.268,Z 837.512,A -85,B 0,C 180,E1 -19323.79,E2 -19323.79} C_VEL
LIN {X 0,Y 256.719,Z 849.077,A -85,B 0,C 180,E1 -19325.113,E2 -19325.113} C_VEL
LIN {X 0,Y 254.926,Z 859.535,A -85,B 0,C 180,E1 -19326.643,E2 -19326.643} C_VEL
LIN {X 0,Y 253.03,Z 869.126,A -85,B 0,C 180,E1 -19328.396,E2 -19328.396} C_VEL
LIN {X 0,Y 251.225,Z 877.816,A -85,B 0,C 180,E1 -19330.375,E2 -19330.375} C_VEL
LIN {X 0,Y 249.077,Z 886.315,A -85,B 0,C 180,E1 -19332.756,E2 -19332.756} C_VEL
LIN {X 0,Y 247.241,Z 893.073,A -85,B 0,C 180,E1 -19335.167,E2 -19335.167} C_VEL
LIN {X 0,Y 245.994,Z 898.435,A -85,B 0,C 180,E1 -19337.617,E2 -19337.617} C_VEL
LIN {X 0,Y 245.223,Z 901.37,A -85,B 0,C 180,E1 -19339.253,E2 -19339.253} C_VEL
LIN {X 0,Y 243.929,Z 904.928,A -85,B 0,C 180,E1 -19341.707,E2 -19341.707} C_VEL
LIN {X 0,Y 243.37,Z 906.75,A -85,B 0,C 180,E1 -19343.356,E2 -19343.356} C_VEL
LIN {X 0,Y 242.918,Z 909.057,A -85,B 0,C 180,E1 -19346.672,E2 -19346.672} C_VEL
LIN {X 0,Y 242.612,Z 909.896,A -85,B 0,C 180,E1 -19349.989,E2 -19349.989} C_VEL
LIN {X 0,Y 242.912,Z 909.129,A -85,B 0,C 180,E1 -19353.306,E2 -19353.306} C_VEL
LIN {X 0,Y 243.348,Z 906.897,A -85,B 0,C 180,E1 -19356.622,E2 -19356.622} C_VEL
LIN {X 0,Y 244.28,Z 904.076,A -85,B 0,C 180,E1 -19359.093,E2 -19359.093} C_VEL
LIN {X 0,Y 245.525,Z 900.246,A -85,B 0,C 180,E1 -19361.547,E2 -19361.547} C_VEL
LIN {X 0,Y 246.912,Z 894.77,A -85,B 0,C 180,E1 -19364.25,E2 -19364.25} C_VEL
LIN {X 0,Y 248.716,Z 887.954,A -85,B 0,C 180,E1 -19366.824,E2 -19366.824} C_VEL
LIN {X 0,Y 250.788,Z 879.921,A -85,B 0,C 180,E1 -19369.212,E2 -19369.212} C_VEL
LIN {X 0,Y 252.627,Z 871.697,A -85,B 0,C 180,E1 -19371.189,E2 -19371.189} C_VEL
LIN {X 0,Y 254.615,Z 861.519,A -85,B 0,C 180,E1 -19373.149,E2 -19373.149} C_VEL
LIN {X 0,Y 256.522,Z 851.041,A -85,B 0,C 180,E1 -19374.739,E2 -19374.739} C_VEL
LIN {X 0,Y 258.151,Z 839.762,A -85,B 0,C 180,E1 -19376.096,E2 -19376.096} C_VEL
LIN {X 0,Y 259.501,Z 827.809,A -85,B 0,C 180,E1 -19377.181,E2 -19377.181} C_VEL
LIN {X 0,Y 260.16,Z 814.87,A -85,B 0,C 180,E1 -19378.061,E2 -19378.061} C_VEL
LIN {X 0,Y 260.51,Z 802.17,A -85,B 0,C 180,E1 -19378.607,E2 -19378.607} C_VEL
LIN {X 0,Y 261.44,Z 759.98,A -85,B 0,C 180,E1 -19379.806,E2 -19379.806} C_VEL
LIN {X 0,Y 254.439,Z 745.282,A -85,B 0,C 180,E1 -19381.229,E2 -19381.229} C_VEL
LIN {X 0,Y 247.097,Z 732.041,A -85,B 0,C 180,E1 -19382.759,E2 -19382.759} C_VEL
LIN {X 0,Y 243.495,Z 725.876,A -85,B 0,C 180,E1 -19383.543,E2 -19383.543} C_VEL
LIN {X 0,Y 242.225,Z 723.424,A -85,B 0,C 180,E1 -19383.837,E2 -19383.837} C_VEL
LIN {X 0,Y 241.989,Z 722.339,A -85,B 0,C 180,E1 -19383.949,E2 -19383.949} C_VEL
LIN {X 0,Y 241.985,Z 722.32,A -85,B 0,C 180,E1 -19388.356,E2 -19388.356} C_VEL
LIN {X 0,Y 241.999,Z 722.346,A -85,B 0,C 180,E1 -19391.891,E2 -19391.891} C_VEL
LIN {X 0,Y 241.982,Z 722.322,A -85,B 0,C 180,E1 -19396.539,E2 -19396.539} C_VEL
LIN {X 0,Y 241.965,Z 722.341,A -85,B 0,C 180,E1 -19400.282,E2 -19400.282} C_VEL
LIN {X 0,Y 241.989,Z 722.338,A -85,B 0,C 180,E1 -19404.489,E2 -19404.489} C_VEL
LIN {X 0,Y 241.923,Z 722.349,A -85,B 0,C 180,E1 -19408.472,E2 -19408.472} C_VEL
LIN {X 0,Y 241.946,Z 722.34,A -85,B 0,C 180,E1 -19412.305,E2 -19412.305} C_VEL
LIN {X 0,Y 241.984,Z 722.33,A -85,B 0,C 180,E1 -19416.008,E2 -19416.008} C_VEL
LIN {X 0,Y 241.977,Z 722.343,A -85,B 0,C 180,E1 -19419.602,E2 -19419.602} C_VEL
LIN {X 0,Y 242.104,Z 722.313,A -85,B 0,C 180,E1 -19423.274,E2 -19423.274} C_VEL
LIN {X 0,Y 242.123,Z 722.314,A -85,B 0,C 180,E1 -19428.277,E2 -19428.277} C_VEL
LIN {X 0,Y 242.351,Z 722.298,A -85,B 0,C 180,E1 -19431.663,E2 -19431.663} C_VEL
LIN {X 0,Y 242.201,Z 722.306,A -85,B 0,C 180,E1 -19435.006,E2 -19435.006} C_VEL
LIN {X 0,Y 242.581,Z 722.269,A -85,B 0,C 180,E1 -19438.34,E2 -19438.34} C_VEL
LIN {X 0,Y 242.581,Z 722.262,A -85,B 0,C 180,E1 -19441.66,E2 -19441.66} C_VEL
LIN {X 0,Y 242.233,Z 722.304,A -85,B 0,C 180,E1 -19444.302,E2 -19444.302} C_VEL
LIN {X 0,Y 241.504,Z 722.407,A -85,B 0,C 180,E1 -19445.691,E2 -19445.691} C_VEL
LIN {X 0,Y 238.626,Z 722.755,A -85,B 0,C 180,E1 -19447.957,E2 -19447.957} C_VEL
LIN {X 0,Y 236.206,Z 723.052,A -85,B 0,C 180,E1 -19449.803,E2 -19449.803} C_VEL
LIN {X 0,Y 235.156,Z 723.191,A -85,B 0,C 180,E1 -19451.235,E2 -19451.235} C_VEL
LIN {X 0,Y 235.061,Z 723.202,A -85,B 0,C 180,E1 -19451.721,E2 -19451.721} C_VEL
LIN {X 0,Y 235.042,Z 723.207,A -85,B 0,C 180,E1 -19455.611,E2 -19455.611} C_VEL
LIN {X 0,Y 234.946,Z 723.214,A -85,B 0,C 180,E1 -19459.211,E2 -19459.211} C_VEL
LIN {X 0,Y 234.903,Z 723.222,A -85,B 0,C 180,E1 -19462.889,E2 -19462.889} C_VEL
LIN {X 0,Y 234.913,Z 723.212,A -85,B 0,C 180,E1 -19466.664,E2 -19466.664} C_VEL
LIN {X 0,Y 234.87,Z 723.217,A -85,B 0,C 180,E1 -19470.577,E2 -19470.577} C_VEL
LIN {X 0,Y 234.911,Z 723.216,A -85,B 0,C 180,E1 -19474.641,E2 -19474.641} C_VEL
LIN {X 0,Y 234.921,Z 723.197,A -85,B 0,C 180,E1 -19478.961,E2 -19478.961} C_VEL
LIN {X 0,Y 234.971,Z 723.317,A -85,B 0,C 180,E1 -19482.333,E2 -19482.333} C_VEL
LIN {X 0,Y 238.177,Z 734.545,A -85,B 0,C 180,E1 -19486.862,E2 -19486.862} C_VEL
LIN {X 0,Y 240.398,Z 742.985,A -85,B 0,C 180,E1 -19489.99,E2 -19489.99} C_VEL
LIN {X 0,Y 242.587,Z 753.001,A -85,B 0,C 180,E1 -19493.441,E2 -19493.441} C_VEL
LIN {X 0,Y 243.998,Z 760.102,A -85,B 0,C 180,E1 -19495.766,E2 -19495.766} C_VEL
LIN {X 0,Y 245.292,Z 764.425,A -85,B 0,C 180,E1 -19496.111,E2 -19496.111} C_VEL
LIN {X 0,Y 248.852,Z 791.487,A -85,B 0,C 180,E1 -19497.541,E2 -19497.541} C_VEL
LIN {X 0,Y 251.903,Z 824.277,A -85,B 0,C 180,E1 -19499.028,E2 -19499.028} C_VEL
LIN {X 0,Y 252.869,Z 838.901,A -85,B 0,C 180,E1 -19499.623,E2 -19499.623} C_VEL
LIN {X 0,Y 251.553,Z 873.024,A -85,B 0,C 180,E1 -19500.613,E2 -19500.613} C_VEL
LIN {X 0,Y 250.234,Z 886.804,A -85,B 0,C 180,E1 -19501.32,E2 -19501.32} C_VEL
LIN {X 0,Y 248.508,Z 899.556,A -85,B 0,C 180,E1 -19502.313,E2 -19502.313} C_VEL
LIN {X 0,Y 246.343,Z 911.285,A -85,B 0,C 180,E1 -19503.541,E2 -19503.541} C_VEL
LIN {X 0,Y 243.88,Z 922.631,A -85,B 0,C 180,E1 -19505.087,E2 -19505.087} C_VEL
LIN {X 0,Y 241.477,Z 932.899,A -85,B 0,C 180,E1 -19506.878,E2 -19506.878} C_VEL
LIN {X 0,Y 239.167,Z 942.184,A -85,B 0,C 180,E1 -19508.915,E2 -19508.915} C_VEL
LIN {X 0,Y 237.142,Z 951.059,A -85,B 0,C 180,E1 -19511.356,E2 -19511.356} C_VEL
LIN {X 0,Y 235.702,Z 957.539,A -85,B 0,C 180,E1 -19513.558,E2 -19513.558} C_VEL
LIN {X 0,Y 234.524,Z 963.709,A -85,B 0,C 180,E1 -19516.142,E2 -19516.142} C_VEL
LIN {X 0,Y 233.892,Z 968.64,A -85,B 0,C 180,E1 -19518.749,E2 -19518.749} C_VEL
LIN {X 0,Y 233.774,Z 972.47,A -85,B 0,C 180,E1 -19521.367,E2 -19521.367} C_VEL
LIN {X 0,Y 233.925,Z 974.473,A -85,B 0,C 180,E1 -19523.11,E2 -19523.11} C_VEL
LIN {X 0,Y 234.155,Z 975.992,A -85,B 0,C 180,E1 -19524.846,E2 -19524.846} C_VEL
LIN {X 0,Y 234.384,Z 977.084,A -85,B 0,C 180,E1 -19526.574,E2 -19526.574} C_VEL
LIN {X 0,Y 234.591,Z 977.757,A -85,B 0,C 180,E1 -19528.295,E2 -19528.295} C_VEL
LIN {X 0,Y 234.808,Z 978.009,A -85,B 0,C 180,E1 -19530.011,E2 -19530.011} C_VEL
LIN {X 0,Y 234.589,Z 977.74,A -85,B 0,C 180,E1 -19531.728,E2 -19531.728} C_VEL
LIN {X 0,Y 234.38,Z 977.054,A -85,B 0,C 180,E1 -19533.449,E2 -19533.449} C_VEL
LIN {X 0,Y 234.122,Z 975.946,A -85,B 0,C 180,E1 -19535.178,E2 -19535.178} C_VEL
LIN {X 0,Y 233.842,Z 973.937,A -85,B 0,C 180,E1 -19537.342,E2 -19537.342} C_VEL
LIN {X 0,Y 233.806,Z 970.653,A -85,B 0,C 180,E1 -19540.401,E2 -19540.401} C_VEL
LIN {X 0,Y 234.525,Z 967.448,A -85,B 0,C 180,E1 -19543.882,E2 -19543.882} C_VEL
LIN {X 0,Y 236.188,Z 962.604,A -85,B 0,C 180,E1 -19547.322,E2 -19547.322} C_VEL
LIN {X 0,Y 238.391,Z 957.963,A -85,B 0,C 180,E1 -19549.828,E2 -19549.828} C_VEL
LIN {X 0,Y 241.614,Z 951.167,A -85,B 0,C 180,E1 -19552.68,E2 -19552.68} C_VEL
LIN {X 0,Y 245.048,Z 944.158,A -85,B 0,C 180,E1 -19555.036,E2 -19555.036} C_VEL
LIN {X 0,Y 249.31,Z 935.779,A -85,B 0,C 180,E1 -19557.274,E2 -19557.274} C_VEL
LIN {X 0,Y 253.245,Z 927.631,A -85,B 0,C 180,E1 -19559.065,E2 -19559.065} C_VEL
LIN {X 0,Y 257.702,Z 918.076,A -85,B 0,C 180,E1 -19560.763,E2 -19560.763} C_VEL
LIN {X 0,Y 261.582,Z 909.248,A -85,B 0,C 180,E1 -19562.057,E2 -19562.057} C_VEL
LIN {X 0,Y 265.757,Z 898.904,A -85,B 0,C 180,E1 -19563.29,E2 -19563.29} C_VEL
LIN {X 0,Y 269.602,Z 888.434,A -85,B 0,C 180,E1 -19564.323,E2 -19564.323} C_VEL
LIN {X 0,Y 273.163,Z 877.611,A -85,B 0,C 180,E1 -19565.156,E2 -19565.156} C_VEL
LIN {X 0,Y 276.967,Z 863.533,A -85,B 0,C 180,E1 -19566.051,E2 -19566.051} C_VEL
LIN {X 0,Y 280.562,Z 845.492,A -85,B 0,C 180,E1 -19566.964,E2 -19566.964} C_VEL
LIN {X 0,Y 282.863,Z 827.718,A -85,B 0,C 180,E1 -19568.242,E2 -19568.242} C_VEL
LIN {X 0,Y 284.51,Z 813.073,A -85,B 0,C 180,E1 -19569.604,E2 -19569.604} C_VEL
LIN {X 0,Y 286.496,Z 796.88,A -85,B 0,C 180,E1 -19571.357,E2 -19571.357} C_VEL
LIN {X 0,Y 286.745,Z 794.701,A -85,B 0,C 180,E1 -19571.672,E2 -19571.672} C_VEL
LIN {X 0,Y 287.045,Z 787.133,A -85,B 0,C 180,E1 -19573.711,E2 -19573.711} C_VEL
LIN {X 0,Y 286.734,Z 785.908,A -85,B 0,C 180,E1 -19575.085,E2 -19575.085} C_VEL
LIN {X 0,Y 286.728,Z 785.399,A -85,B 0,C 180,E1 -19577.344,E2 -19577.344} C_VEL
LIN {X 0,Y 287.579,Z 785.752,A -85,B 0,C 180,E1 -19579.598,E2 -19579.598} C_VEL
LIN {X 0,Y 288.451,Z 786.592,A -85,B 0,C 180,E1 -19580.906,E2 -19580.906} C_VEL
LIN {X 0,Y 289.719,Z 790.166,A -85,B 0,C 180,E1 -19582.772,E2 -19582.772} C_VEL
LIN {X 0,Y 289.811,Z 790.486,A -85,B 0,C 180,E1 -19582.888,E2 -19582.888} C_VEL
LIN {X 0,Y 284.972,Z 816.766,A -85,B 0,C 180,E1 -19584.249,E2 -19584.249} C_VEL
LIN {X 0,Y 282.541,Z 831.288,A -85,B 0,C 180,E1 -19585.211,E2 -19585.211} C_VEL
LIN {X 0,Y 280.224,Z 842.048,A -85,B 0,C 180,E1 -19586.08,E2 -19586.08} C_VEL
LIN {X 0,Y 276.471,Z 855.789,A -85,B 0,C 180,E1 -19587.52,E2 -19587.52} C_VEL
LIN {X 0,Y 273.401,Z 864.991,A -85,B 0,C 180,E1 -19588.739,E2 -19588.739} C_VEL
LIN {X 0,Y 269.559,Z 874.74,A -85,B 0,C 180,E1 -19590.306,E2 -19590.306} C_VEL
LIN {X 0,Y 266.492,Z 881.695,A -85,B 0,C 180,E1 -19591.66,E2 -19591.66} C_VEL
LIN {X 0,Y 262.838,Z 889.024,A -85,B 0,C 180,E1 -19593.392,E2 -19593.392} C_VEL
LIN {X 0,Y 259.333,Z 895.259,A -85,B 0,C 180,E1 -19595.162,E2 -19595.162} C_VEL
LIN {X 0,Y 256.708,Z 899.454,A -85,B 0,C 180,E1 -19596.611,E2 -19596.611} C_VEL
LIN {X 0,Y 252.993,Z 904.709,A -85,B 0,C 180,E1 -19598.83,E2 -19598.83} C_VEL
LIN {X 0,Y 249.612,Z 908.766,A -85,B 0,C 180,E1 -19601.108,E2 -19601.108} C_VEL
LIN {X 0,Y 246.546,Z 911.782,A -85,B 0,C 180,E1 -19603.438,E2 -19603.438} C_VEL
LIN {X 0,Y 244.753,Z 913.258,A -85,B 0,C 180,E1 -19605.023,E2 -19605.023} C_VEL
LIN {X 0,Y 243.031,Z 914.281,A -85,B 0,C 180,E1 -19606.624,E2 -19606.624} C_VEL
LIN {X 0,Y 240.089,Z 915.049,A -85,B 0,C 180,E1 -19609.884,E2 -19609.884} C_VEL
LIN {X 0,Y 238.979,Z 914.77,A -85,B 0,C 180,E1 -19611.544,E2 -19611.544} C_VEL
LIN {X 0,Y 237.994,Z 914.092,A -85,B 0,C 180,E1 -19613.216,E2 -19613.216} C_VEL
LIN {X 0,Y 237.283,Z 912.947,A -85,B 0,C 180,E1 -19614.902,E2 -19614.902} C_VEL
LIN {X 0,Y 236.202,Z 910.488,A -85,B 0,C 180,E1 -19617.442,E2 -19617.442} C_VEL
LIN {X 0,Y 235.372,Z 907.004,A -85,B 0,C 180,E1 -19620,E2 -19620} C_VEL
LIN {X 0,Y 235.002,Z 902.423,A -85,B 0,C 180,E1 -19622.571,E2 -19622.571} C_VEL
LIN {X 0,Y 234.897,Z 896.644,A -85,B 0,C 180,E1 -19625.15,E2 -19625.15} C_VEL
LIN {X 0,Y 235.245,Z 890.846,A -85,B 0,C 180,E1 -19627.295,E2 -19627.295} C_VEL
LIN {X 0,Y 235.594,Z 884.24,A -85,B 0,C 180,E1 -19629.35,E2 -19629.35} C_VEL
LIN {X 0,Y 236.107,Z 875.808,A -85,B 0,C 180,E1 -19631.547,E2 -19631.547} C_VEL
LIN {X 0,Y 236.763,Z 866.795,A -85,B 0,C 180,E1 -19633.519,E2 -19633.519} C_VEL
LIN {X 0,Y 237.414,Z 857.513,A -85,B 0,C 180,E1 -19635.232,E2 -19635.232} C_VEL
LIN {X 0,Y 238.036,Z 847.884,A -85,B 0,C 180,E1 -19636.731,E2 -19636.731} C_VEL
LIN {X 0,Y 238.742,Z 838.102,A -85,B 0,C 180,E1 -19638.005,E2 -19638.005} C_VEL
LIN {X 0,Y 239.4,Z 826.602,A -85,B 0,C 180,E1 -19639.237,E2 -19639.237} C_VEL
LIN {X 0,Y 239.998,Z 812.31,A -85,B 0,C 180,E1 -19640.413,E2 -19640.413} C_VEL
LIN {X 0,Y 240.373,Z 796.947,A -85,B 0,C 180,E1 -19641.268,E2 -19641.268} C_VEL
LIN {X 0,Y 241.921,Z 746.948,A -85,B 0,C 180,E1 -19643.589,E2 -19643.589} C_VEL
LIN {X 0,Y 235.06,Z 723.203,A -85,B 0,C 180,E1 -19645.099,E2 -19645.099} C_VEL
LIN {X 0,Y 234.922,Z 723.22,A -85,B 0,C 180,E1 -19650.569,E2 -19650.569} C_VEL
LIN {X 0,Y 234.949,Z 723.217,A -85,B 0,C 180,E1 -19654.635,E2 -19654.635} C_VEL
LIN {X 0,Y 234.939,Z 723.215,A -85,B 0,C 180,E1 -19658.93,E2 -19658.93} C_VEL
LIN {X 0,Y 234.877,Z 723.221,A -85,B 0,C 180,E1 -19663.489,E2 -19663.489} C_VEL
LIN {X 0,Y 234.876,Z 723.219,A -85,B 0,C 180,E1 -19666.5,E2 -19666.5} C_VEL
LIN {X 0,Y 234.941,Z 723.211,A -85,B 0,C 180,E1 -19671.072,E2 -19671.072} C_VEL
LIN {X 0,Y 234.978,Z 723.383,A -85,B 0,C 180,E1 -19675.072,E2 -19675.072} C_VEL
LIN {X 0,Y 235.994,Z 726.134,A -85,B 0,C 180,E1 -19675.352,E2 -19675.352} C_VEL
LIN {X 0,Y 237.59,Z 728.495,A -85,B 0,C 180,E1 -19675.714,E2 -19675.714} C_VEL
LIN {X 0,Y 246.218,Z 743.604,A -85,B 0,C 180,E1 -19677.642,E2 -19677.642} C_VEL
LIN {X 0,Y 254.259,Z 759.732,A -85,B 0,C 180,E1 -19679.354,E2 -19679.354} C_VEL
LIN {X 0,Y 255.293,Z 762.119,A -85,B 0,C 180,E1 -19679.574,E2 -19679.574} C_VEL
LIN {X 0,Y 254.353,Z 796.338,A -85,B 0,C 180,E1 -19680.549,E2 -19680.549} C_VEL
LIN {X 0,Y 254.041,Z 812.422,A -85,B 0,C 180,E1 -19681.136,E2 -19681.136} C_VEL
LIN {X 0,Y 253.426,Z 824.422,A -85,B 0,C 180,E1 -19681.862,E2 -19681.862} C_VEL
LIN {X 0,Y 252.112,Z 837.444,A -85,B 0,C 180,E1 -19682.976,E2 -19682.976} C_VEL
LIN {X 0,Y 250.562,Z 848.948,A -85,B 0,C 180,E1 -19684.295,E2 -19684.295} C_VEL
LIN {X 0,Y 248.67,Z 859.374,A -85,B 0,C 180,E1 -19685.797,E2 -19685.797} C_VEL
LIN {X 0,Y 246.951,Z 868.199,A -85,B 0,C 180,E1 -19687.396,E2 -19687.396} C_VEL
LIN {X 0,Y 244.996,Z 877.231,A -85,B 0,C 180,E1 -19689.417,E2 -19689.417} C_VEL
LIN {X 0,Y 242.703,Z 886.011,A -85,B 0,C 180,E1 -19691.853,E2 -19691.853} C_VEL
LIN {X 0,Y 240.595,Z 893.677,A -85,B 0,C 180,E1 -19694.572,E2 -19694.572} C_VEL
LIN {X 0,Y 239.134,Z 899.439,A -85,B 0,C 180,E1 -19697.256,E2 -19697.256} C_VEL
LIN {X 0,Y 238.322,Z 902.373,A -85,B 0,C 180,E1 -19698.938,E2 -19698.938} C_VEL
LIN {X 0,Y 236.977,Z 905.931,A -85,B 0,C 180,E1 -19701.462,E2 -19701.462} C_VEL
LIN {X 0,Y 236.39,Z 907.753,A -85,B 0,C 180,E1 -19703.159,E2 -19703.159} C_VEL
LIN {X 0,Y 235.902,Z 910.06,A -85,B 0,C 180,E1 -19706.573,E2 -19706.573} C_VEL
LIN {X 0,Y 235.584,Z 910.898,A -85,B 0,C 180,E1 -19709.989,E2 -19709.989} C_VEL
LIN {X 0,Y 235.896,Z 910.131,A -85,B 0,C 180,E1 -19713.404,E2 -19713.404} C_VEL
LIN {X 0,Y 236.368,Z 907.899,A -85,B 0,C 180,E1 -19716.819,E2 -19716.819} C_VEL
LIN {X 0,Y 237.344,Z 905.077,A -85,B 0,C 180,E1 -19719.361,E2 -19719.361} C_VEL
LIN {X 0,Y 238.644,Z 901.248,A -85,B 0,C 180,E1 -19721.884,E2 -19721.884} C_VEL
LIN {X 0,Y 240.106,Z 895.771,A -85,B 0,C 180,E1 -19724.663,E2 -19724.663} C_VEL
LIN {X 0,Y 241.997,Z 888.954,A -85,B 0,C 180,E1 -19727.305,E2 -19727.305} C_VEL
LIN {X 0,Y 244.163,Z 880.921,A -85,B 0,C 180,E1 -19729.755,E2 -19729.755} C_VEL
LIN {X 0,Y 246.087,Z 872.697,A -85,B 0,C 180,E1 -19731.78,E2 -19731.78} C_VEL
LIN {X 0,Y 248.167,Z 862.518,A -85,B 0,C 180,E1 -19733.787,E2 -19733.787} C_VEL
LIN {X 0,Y 250.152,Z 852.04,A -85,B 0,C 180,E1 -19735.413,E2 -19735.413} C_VEL
LIN {X 0,Y 251.858,Z 840.759,A -85,B 0,C 180,E1 -19736.8,E2 -19736.8} C_VEL
LIN {X 0,Y 253.269,Z 828.803,A -85,B 0,C 180,E1 -19737.908,E2 -19737.908} C_VEL
LIN {X 0,Y 253.981,Z 815.545,A -85,B 0,C 180,E1 -19738.827,E2 -19738.827} C_VEL
LIN {X 0,Y 254.345,Z 803.155,A -85,B 0,C 180,E1 -19739.367,E2 -19739.367} C_VEL
LIN {X 0,Y 255.282,Z 762.021,A -85,B 0,C 180,E1 -19740.567,E2 -19740.567} C_VEL
LIN {X 0,Y 248.778,Z 748.367,A -85,B 0,C 180,E1 -19741.95,E2 -19741.95} C_VEL
LIN {X 0,Y 240.772,Z 733.926,A -85,B 0,C 180,E1 -19743.704,E2 -19743.704} C_VEL
LIN {X 0,Y 236.628,Z 726.978,A -85,B 0,C 180,E1 -19744.655,E2 -19744.655} C_VEL
LIN {X 0,Y 235.275,Z 724.631,A -85,B 0,C 180,E1 -19744.978,E2 -19744.978} C_VEL
LIN {X 0,Y 234.962,Z 723.216,A -85,B 0,C 180,E1 -19745.136,E2 -19745.136} C_VEL
LIN {X 0,Y 234.933,Z 723.2,A -85,B 0,C 180,E1 -19748.941,E2 -19748.941} C_VEL
LIN {X 0,Y 234.957,Z 723.202,A -85,B 0,C 180,E1 -19753.45,E2 -19753.45} C_VEL
LIN {X 0,Y 234.954,Z 723.197,A -85,B 0,C 180,E1 -19756.529,E2 -19756.529} C_VEL
LIN {X 0,Y 234.91,Z 723.216,A -85,B 0,C 180,E1 -19761.077,E2 -19761.077} C_VEL
LIN {X 0,Y 234.912,Z 723.214,A -85,B 0,C 180,E1 -19765.359,E2 -19765.359} C_VEL
LIN {X 0,Y 234.871,Z 723.224,A -85,B 0,C 180,E1 -19769.423,E2 -19769.423} C_VEL
LIN {X 0,Y 234.939,Z 723.22,A -85,B 0,C 180,E1 -19773.788,E2 -19773.788} C_VEL
LIN {X 0,Y 234.94,Z 723.22,A -85,B 0,C 180,E1 -19778.963,E2 -19778.963} C_VEL
LIN {X 0,Y 235.037,Z 723.192,A -85,B 0,C 180,E1 -19783.056,E2 -19783.056} C_VEL
LIN {X 0,Y 235.055,Z 723.198,A -85,B 0,C 180,E1 -19787.919,E2 -19787.919} C_VEL
LIN {X 0,Y 235.283,Z 723.177,A -85,B 0,C 180,E1 -19791.41,E2 -19791.41} C_VEL
LIN {X 0,Y 235.335,Z 723.174,A -85,B 0,C 180,E1 -19793.139,E2 -19793.139} C_VEL
LIN {X 0,Y 235.541,Z 723.146,A -85,B 0,C 180,E1 -19798.29,E2 -19798.29} C_VEL
LIN {X 0,Y 235.541,Z 723.138,A -85,B 0,C 180,E1 -19801.71,E2 -19801.71} C_VEL
LIN {X 0,Y 235.335,Z 723.173,A -85,B 0,C 180,E1 -19806.861,E2 -19806.861} C_VEL
LIN {X 0,Y 235.176,Z 723.182,A -85,B 0,C 180,E1 -19810.329,E2 -19810.329} C_VEL
LIN {X 0,Y 235.061,Z 723.202,A -85,B 0,C 180,E1 -19811.721,E2 -19811.721} C_VEL
LIN {X 0,Y 234.356,Z 723.3,A -85,B 0,C 180,E1 -19813.151,E2 -19813.151} C_VEL
LIN {X 0,Y 231.45,Z 723.662,A -85,B 0,C 180,E1 -19815.483,E2 -19815.483} C_VEL
LIN {X 0,Y 229,Z 723.958,A -85,B 0,C 180,E1 -19817.385,E2 -19817.385} C_VEL
LIN {X 0,Y 227.956,Z 724.089,A -85,B 0,C 180,E1 -19818.862,E2 -19818.862} C_VEL
LIN {X 0,Y 227.874,Z 724.089,A -85,B 0,C 180,E1 -19819.363,E2 -19819.363} C_VEL
LIN {X 0,Y 227.856,Z 724.103,A -85,B 0,C 180,E1 -19823.639,E2 -19823.639} C_VEL
LIN {X 0,Y 227.825,Z 724.101,A -85,B 0,C 180,E1 -19827.563,E2 -19827.563} C_VEL
LIN {X 0,Y 227.817,Z 724.102,A -85,B 0,C 180,E1 -19831.63,E2 -19831.63} C_VEL
LIN {X 0,Y 227.853,Z 724.104,A -85,B 0,C 180,E1 -19835.877,E2 -19835.877} C_VEL
LIN {X 0,Y 227.88,Z 724.105,A -85,B 0,C 180,E1 -19841.167,E2 -19841.167} C_VEL
LIN {X 0,Y 230.92,Z 734.478,A -85,B 0,C 180,E1 -19845.593,E2 -19845.593} C_VEL
LIN {X 0,Y 233.534,Z 744.306,A -85,B 0,C 180,E1 -19849.412,E2 -19849.412} C_VEL
LIN {X 0,Y 236.008,Z 755.808,A -85,B 0,C 180,E1 -19853.516,E2 -19853.516} C_VEL
LIN {X 0,Y 236.684,Z 759.076,A -85,B 0,C 180,E1 -19854.56,E2 -19854.56} C_VEL
LIN {X 0,Y 239.451,Z 766.248,A -85,B 0,C 180,E1 -19855.267,E2 -19855.267} C_VEL
LIN {X 0,Y 242.957,Z 793.826,A -85,B 0,C 180,E1 -19856.766,E2 -19856.766} C_VEL
LIN {X 0,Y 245.795,Z 825.542,A -85,B 0,C 180,E1 -19858.245,E2 -19858.245} C_VEL
LIN {X 0,Y 246.654,Z 840.478,A -85,B 0,C 180,E1 -19858.858,E2 -19858.858} C_VEL
LIN {X 0,Y 245.397,Z 871.271,A -85,B 0,C 180,E1 -19859.762,E2 -19859.762} C_VEL
LIN {X 0,Y 244.06,Z 885.342,A -85,B 0,C 180,E1 -19860.489,E2 -19860.489} C_VEL
LIN {X 0,Y 242.424,Z 897.539,A -85,B 0,C 180,E1 -19861.437,E2 -19861.437} C_VEL
LIN {X 0,Y 240.31,Z 908.68,A -85,B 0,C 180,E1 -19862.588,E2 -19862.588} C_VEL
LIN {X 0,Y 237.787,Z 920.323,A -85,B 0,C 180,E1 -19864.169,E2 -19864.169} C_VEL
LIN {X 0,Y 235.223,Z 930.837,A -85,B 0,C 180,E1 -19865.992,E2 -19865.992} C_VEL
LIN {X 0,Y 232.95,Z 939.465,A -85,B 0,C 180,E1 -19867.859,E2 -19867.859} C_VEL
LIN {X 0,Y 230.95,Z 947.48,A -85,B 0,C 180,E1 -19869.994,E2 -19869.994} C_VEL
LIN {X 0,Y 229.015,Z 955.352,A -85,B 0,C 180,E1 -19872.603,E2 -19872.603} C_VEL
LIN {X 0,Y 227.581,Z 962.689,A -85,B 0,C 180,E1 -19875.71,E2 -19875.71} C_VEL
LIN {X 0,Y 226.886,Z 967.621,A -85,B 0,C 180,E1 -19878.397,E2 -19878.397} C_VEL
LIN {X 0,Y 226.701,Z 971.45,A -85,B 0,C 180,E1 -19881.095,E2 -19881.095} C_VEL
LIN {X 0,Y 226.833,Z 973.454,A -85,B 0,C 180,E1 -19882.893,E2 -19882.893} C_VEL
LIN {X 0,Y 227.073,Z 974.978,A -85,B 0,C 180,E1 -19884.685,E2 -19884.685} C_VEL
LIN {X 0,Y 227.329,Z 976.076,A -85,B 0,C 180,E1 -19886.467,E2 -19886.467} C_VEL
LIN {X 0,Y 227.54,Z 976.75,A -85,B 0,C 180,E1 -19888.242,E2 -19888.242} C_VEL
LIN {X 0,Y 227.771,Z 977.005,A -85,B 0,C 180,E1 -19890.012,E2 -19890.012} C_VEL
LIN {X 0,Y 227.537,Z 976.733,A -85,B 0,C 180,E1 -19891.782,E2 -19891.782} C_VEL
LIN {X 0,Y 227.322,Z 976.045,A -85,B 0,C 180,E1 -19893.557,E2 -19893.557} C_VEL
LIN {X 0,Y 227.041,Z 974.931,A -85,B 0,C 180,E1 -19895.34,E2 -19895.34} C_VEL
LIN {X 0,Y 226.775,Z 973.126,A -85,B 0,C 180,E1 -19897.379,E2 -19897.379} C_VEL
LIN {X 0,Y 226.797,Z 969.656,A -85,B 0,C 180,E1 -19900.727,E2 -19900.727} C_VEL
LIN {X 0,Y 227.053,Z 968.36,A -85,B 0,C 180,E1 -19902.525,E2 -19902.525} C_VEL
LIN {X 0,Y 228.33,Z 964.612,A -85,B 0,C 180,E1 -19906.093,E2 -19906.093} C_VEL
LIN {X 0,Y 229.998,Z 960.912,A -85,B 0,C 180,E1 -19908.691,E2 -19908.691} C_VEL
LIN {X 0,Y 232.584,Z 956.192,A -85,B 0,C 180,E1 -19911.271,E2 -19911.271} C_VEL
LIN {X 0,Y 236.202,Z 949.39,A -85,B 0,C 180,E1 -19914.16,E2 -19914.16} C_VEL
LIN {X 0,Y 240.092,Z 942.413,A -85,B 0,C 180,E1 -19916.523,E2 -19916.523} C_VEL
LIN {X 0,Y 243.891,Z 935.579,A -85,B 0,C 180,E1 -19918.4,E2 -19918.4} C_VEL
LIN {X 0,Y 248.06,Z 927.761,A -85,B 0,C 180,E1 -19920.202,E2 -19920.202} C_VEL
LIN {X 0,Y 253.216,Z 917.531,A -85,B 0,C 180,E1 -19922.07,E2 -19922.07} C_VEL
LIN {X 0,Y 257.858,Z 907.8,A -85,B 0,C 180,E1 -19923.509,E2 -19923.509} C_VEL
LIN {X 0,Y 262.257,Z 897.647,A -85,B 0,C 180,E1 -19924.722,E2 -19924.722} C_VEL
LIN {X 0,Y 266.905,Z 885.681,A -85,B 0,C 180,E1 -19925.874,E2 -19925.874} C_VEL
LIN {X 0,Y 271.71,Z 871.646,A -85,B 0,C 180,E1 -19926.897,E2 -19926.897} C_VEL
LIN {X 0,Y 275.859,Z 855.527,A -85,B 0,C 180,E1 -19927.818,E2 -19927.818} C_VEL
LIN {X 0,Y 277.867,Z 845.555,A -85,B 0,C 180,E1 -19928.357,E2 -19928.357} C_VEL
LIN {X 0,Y 280.243,Z 829.393,A -85,B 0,C 180,E1 -19929.544,E2 -19929.544} C_VEL
LIN {X 0,Y 282.389,Z 813.879,A -85,B 0,C 180,E1 -19931.029,E2 -19931.029} C_VEL
LIN {X 0,Y 284.581,Z 799.441,A -85,B 0,C 180,E1 -19932.647,E2 -19932.647} C_VEL
LIN {X 0,Y 285.055,Z 793.38,A -85,B 0,C 180,E1 -19934.357,E2 -19934.357} C_VEL
LIN {X 0,Y 284.87,Z 792.551,A -85,B 0,C 180,E1 -19935.69,E2 -19935.69} C_VEL
LIN {X 0,Y 285.215,Z 792.28,A -85,B 0,C 180,E1 -19938.294,E2 -19938.294} C_VEL
LIN {X 0,Y 286.383,Z 793.057,A -85,B 0,C 180,E1 -19940.471,E2 -19940.471} C_VEL
LIN {X 0,Y 287.055,Z 795.277,A -85,B 0,C 180,E1 -19941.72,E2 -19941.72} C_VEL
LIN {X 0,Y 282.052,Z 820.733,A -85,B 0,C 180,E1 -19943.09,E2 -19943.09} C_VEL
LIN {X 0,Y 279.43,Z 834.747,A -85,B 0,C 180,E1 -19944.047,E2 -19944.047} C_VEL
LIN {X 0,Y 276.434,Z 847.002,A -85,B 0,C 180,E1 -19945.108,E2 -19945.108} C_VEL
LIN {X 0,Y 272.866,Z 858.504,A -85,B 0,C 180,E1 -19946.375,E2 -19946.375} C_VEL
LIN {X 0,Y 269.011,Z 868.764,A -85,B 0,C 180,E1 -19947.79,E2 -19947.79} C_VEL
LIN {X 0,Y 265.129,Z 877.851,A -85,B 0,C 180,E1 -19949.318,E2 -19949.318} C_VEL
LIN {X 0,Y 260.318,Z 887.541,A -85,B 0,C 180,E1 -19951.366,E2 -19951.366} C_VEL
LIN {X 0,Y 255.697,Z 895.327,A -85,B 0,C 180,E1 -19953.472,E2 -19953.472} C_VEL
LIN {X 0,Y 252.125,Z 900.687,A -85,B 0,C 180,E1 -19955.284,E2 -19955.284} C_VEL
LIN {X 0,Y 249.445,Z 904.404,A -85,B 0,C 180,E1 -19956.769,E2 -19956.769} C_VEL
LIN {X 0,Y 245.643,Z 908.843,A -85,B 0,C 180,E1 -19959.045,E2 -19959.045} C_VEL
LIN {X 0,Y 242.189,Z 912.237,A -85,B 0,C 180,E1 -19961.385,E2 -19961.385} C_VEL
LIN {X 0,Y 240.048,Z 913.884,A -85,B 0,C 180,E1 -19962.976,E2 -19962.976} C_VEL
LIN {X 0,Y 236.35,Z 915.997,A -85,B 0,C 180,E1 -19966.238,E2 -19966.238} C_VEL
LIN {X 0,Y 233.24,Z 916.402,A -85,B 0,C 180,E1 -19969.584,E2 -19969.584} C_VEL
LIN {X 0,Y 232.074,Z 915.96,A -85,B 0,C 180,E1 -19971.291,E2 -19971.291} C_VEL
LIN {X 0,Y 231.042,Z 915.081,A -85,B 0,C 180,E1 -19973.011,E2 -19973.011} C_VEL
LIN {X 0,Y 229.395,Z 912.114,A -85,B 0,C 180,E1 -19976.487,E2 -19976.487} C_VEL
LIN {X 0,Y 228.59,Z 908.732,A -85,B 0,C 180,E1 -19979.119,E2 -19979.119} C_VEL
LIN {X 0,Y 228.024,Z 904.276,A -85,B 0,C 180,E1 -19981.766,E2 -19981.766} C_VEL
LIN {X 0,Y 227.773,Z 898.594,A -85,B 0,C 180,E1 -19984.424,E2 -19984.424} C_VEL
LIN {X 0,Y 228.109,Z 891.593,A -85,B 0,C 180,E1 -19987.079,E2 -19987.079} C_VEL
LIN {X 0,Y 228.496,Z 884.987,A -85,B 0,C 180,E1 -19989.183,E2 -19989.183} C_VEL
LIN {X 0,Y 228.871,Z 878.11,A -85,B 0,C 180,E1 -19991.065,E2 -19991.065} C_VEL
LIN {X 0,Y 229.477,Z 869.517,A -85,B 0,C 180,E1 -19993.054,E2 -19993.054} C_VEL
LIN {X 0,Y 230.137,Z 860.499,A -85,B 0,C 180,E1 -19994.819,E2 -19994.819} C_VEL
LIN {X 0,Y 230.714,Z 851.181,A -85,B 0,C 180,E1 -19996.366,E2 -19996.366} C_VEL
LIN {X 0,Y 231.428,Z 841.815,A -85,B 0,C 180,E1 -19997.679,E2 -19997.679} C_VEL
LIN {X 0,Y 232.135,Z 830.42,A -85,B 0,C 180,E1 -19998.994,E2 -19998.994} C_VEL
LIN {X 0,Y 232.579,Z 820.462,A -85,B 0,C 180,E1 -19999.927,E2 -19999.927} C_VEL
LIN {X 0,Y 233.022,Z 809.212,A -85,B 0,C 180,E1 -20000.755,E2 -20000.755} C_VEL
LIN {X 0,Y 233.482,Z 791.763,A -85,B 0,C 180,E1 -20001.696,E2 -20001.696} C_VEL
LIN {X 0,Y 234.927,Z 748.287,A -85,B 0,C 180,E1 -20003.821,E2 -20003.821} C_VEL
LIN {X 0,Y 228.088,Z 724.517,A -85,B 0,C 180,E1 -20005.314,E2 -20005.314} C_VEL
LIN {X 0,Y 228.029,Z 724.079,A -85,B 0,C 180,E1 -20005.371,E2 -20005.371} C_VEL
LIN {X 0,Y 227.897,Z 724.096,A -85,B 0,C 180,E1 -20010.274,E2 -20010.274} C_VEL
LIN {X 0,Y 227.903,Z 724.092,A -85,B 0,C 180,E1 -20013.716,E2 -20013.716} C_VEL
LIN {X 0,Y 227.867,Z 724.098,A -85,B 0,C 180,E1 -20018.087,E2 -20018.087} C_VEL
LIN {X 0,Y 227.81,Z 724.104,A -85,B 0,C 180,E1 -20022.743,E2 -20022.743} C_VEL
LIN {X 0,Y 227.809,Z 724.101,A -85,B 0,C 180,E1 -20027.245,E2 -20027.245} C_VEL
LIN {X 0,Y 227.863,Z 724.095,A -85,B 0,C 180,E1 -20031.901,E2 -20031.901} C_VEL
LIN {X 0,Y 227.912,Z 724.087,A -85,B 0,C 180,E1 -20033.78,E2 -20033.78} C_VEL
LIN {X 0,Y 228.972,Z 727.029,A -85,B 0,C 180,E1 -20034.115,E2 -20034.115} C_VEL
LIN {X 0,Y 230.618,Z 729.445,A -85,B 0,C 180,E1 -20034.513,E2 -20034.513} C_VEL
LIN {X 0,Y 238.717,Z 743.247,A -85,B 0,C 180,E1 -20036.435,E2 -20036.435} C_VEL
LIN {X 0,Y 245.727,Z 756.746,A -85,B 0,C 180,E1 -20038.016,E2 -20038.016} C_VEL
LIN {X 0,Y 249.184,Z 764.166,A -85,B 0,C 180,E1 -20038.779,E2 -20038.779} C_VEL
LIN {X 0,Y 248.257,Z 797.365,A -85,B 0,C 180,E1 -20039.752,E2 -20039.752} C_VEL
LIN {X 0,Y 247.905,Z 813.269,A -85,B 0,C 180,E1 -20040.342,E2 -20040.342} C_VEL
LIN {X 0,Y 247.249,Z 825.434,A -85,B 0,C 180,E1 -20041.094,E2 -20041.094} C_VEL
LIN {X 0,Y 245.872,Z 838.454,A -85,B 0,C 180,E1 -20042.232,E2 -20042.232} C_VEL
LIN {X 0,Y 244.248,Z 849.956,A -85,B 0,C 180,E1 -20043.58,E2 -20043.58} C_VEL
LIN {X 0,Y 242.277,Z 860.381,A -85,B 0,C 180,E1 -20045.116,E2 -20045.116} C_VEL
LIN {X 0,Y 240.478,Z 869.205,A -85,B 0,C 180,E1 -20046.752,E2 -20046.752} C_VEL
LIN {X 0,Y 238.43,Z 878.236,A -85,B 0,C 180,E1 -20048.823,E2 -20048.823} C_VEL
LIN {X 0,Y 236.035,Z 887.016,A -85,B 0,C 180,E1 -20051.321,E2 -20051.321} C_VEL
LIN {X 0,Y 233.828,Z 894.682,A -85,B 0,C 180,E1 -20054.114,E2 -20054.114} C_VEL
LIN {X 0,Y 232.285,Z 900.443,A -85,B 0,C 180,E1 -20056.873,E2 -20056.873} C_VEL
LIN {X 0,Y 231.429,Z 903.377,A -85,B 0,C 180,E1 -20058.605,E2 -20058.605} C_VEL
LIN {X 0,Y 230.029,Z 906.935,A -85,B 0,C 180,E1 -20061.202,E2 -20061.202} C_VEL
LIN {X 0,Y 229.413,Z 908.757,A -85,B 0,C 180,E1 -20062.95,E2 -20062.95} C_VEL
LIN {X 0,Y 228.887,Z 911.063,A -85,B 0,C 180,E1 -20066.468,E2 -20066.468} C_VEL
LIN {X 0,Y 228.557,Z 911.901,A -85,B 0,C 180,E1 -20069.988,E2 -20069.988} C_VEL
LIN {X 0,Y 228.881,Z 911.133,A -85,B 0,C 180,E1 -20073.509,E2 -20073.509} C_VEL
LIN {X 0,Y 229.39,Z 908.901,A -85,B 0,C 180,E1 -20077.027,E2 -20077.027} C_VEL
LIN {X 0,Y 230.413,Z 906.079,A -85,B 0,C 180,E1 -20079.645,E2 -20079.645} C_VEL
LIN {X 0,Y 231.771,Z 902.249,A -85,B 0,C 180,E1 -20082.242,E2 -20082.242} C_VEL
LIN {X 0,Y 233.314,Z 896.772,A -85,B 0,C 180,E1 -20085.1,E2 -20085.1} C_VEL
LIN {X 0,Y 235.296,Z 889.955,A -85,B 0,C 180,E1 -20087.814,E2 -20087.814} C_VEL
LIN {X 0,Y 237.56,Z 881.921,A -85,B 0,C 180,E1 -20090.328,E2 -20090.328} C_VEL
LIN {X 0,Y 239.575,Z 873.696,A -85,B 0,C 180,E1 -20092.404,E2 -20092.404} C_VEL
LIN {X 0,Y 241.752,Z 863.517,A -85,B 0,C 180,E1 -20094.459,E2 -20094.459} C_VEL
LIN {X 0,Y 243.822,Z 853.038,A -85,B 0,C 180,E1 -20096.122,E2 -20096.122} C_VEL
LIN {X 0,Y 245.605,Z 841.755,A -85,B 0,C 180,E1 -20097.539,E2 -20097.539} C_VEL
LIN {X 0,Y 247.083,Z 829.796,A -85,B 0,C 180,E1 -20098.67,E2 -20098.67} C_VEL
LIN {X 0,Y 247.836,Z 816.906,A -85,B 0,C 180,E1 -20099.587,E2 -20099.587} C_VEL
LIN {X 0,Y 248.233,Z 803.873,A -85,B 0,C 180,E1 -20100.174,E2 -20100.174} C_VEL
LIN {X 0,Y 249.194,Z 764.016,A -85,B 0,C 180,E1 -20101.363,E2 -20101.363} C_VEL
LIN {X 0,Y 242.315,Z 749.882,A -85,B 0,C 180,E1 -20102.892,E2 -20102.892} C_VEL
LIN {X 0,Y 233.87,Z 734.868,A -85,B 0,C 180,E1 -20104.847,E2 -20104.847} C_VEL
LIN {X 0,Y 229.631,Z 727.915,A -85,B 0,C 180,E1 -20105.881,E2 -20105.881} C_VEL
LIN {X 0,Y 228.149,Z 725.295,A -85,B 0,C 180,E1 -20106.261,E2 -20106.261} C_VEL
LIN {X 0,Y 227.875,Z 724.095,A -85,B 0,C 180,E1 -20106.392,E2 -20106.392} C_VEL
LIN {X 0,Y 227.868,Z 724.095,A -85,B 0,C 180,E1 -20110.349,E2 -20110.349} C_VEL
LIN {X 0,Y 227.88,Z 724.07,A -85,B 0,C 180,E1 -20114.818,E2 -20114.818} C_VEL
LIN {X 0,Y 227.892,Z 724.093,A -85,B 0,C 180,E1 -20117.722,E2 -20117.722} C_VEL
LIN {X 0,Y 227.826,Z 724.1,A -85,B 0,C 180,E1 -20121.905,E2 -20121.905} C_VEL
LIN {X 0,Y 227.84,Z 724.094,A -85,B 0,C 180,E1 -20126.365,E2 -20126.365} C_VEL
LIN {X 0,Y 227.851,Z 724.089,A -85,B 0,C 180,E1 -20130.428,E2 -20130.428} C_VEL
LIN {X 0,Y 227.87,Z 724.097,A -85,B 0,C 180,E1 -20134.419,E2 -20134.419} C_VEL
LIN {X 0,Y 227.891,Z 724.093,A -85,B 0,C 180,E1 -20138.28,E2 -20138.28} C_VEL
LIN {X 0,Y 227.975,Z 724.07,A -85,B 0,C 180,E1 -20142.823,E2 -20142.823} C_VEL
LIN {X 0,Y 228.011,Z 724.08,A -85,B 0,C 180,E1 -20147.54,E2 -20147.54} C_VEL
LIN {X 0,Y 228.219,Z 724.052,A -85,B 0,C 180,E1 -20151.143,E2 -20151.143} C_VEL
LIN {X 0,Y 228.283,Z 724.054,A -85,B 0,C 180,E1 -20152.926,E2 -20152.926} C_VEL
LIN {X 0,Y 228.501,Z 724.023,A -85,B 0,C 180,E1 -20158.237,E2 -20158.237} C_VEL
LIN {X 0,Y 228.501,Z 724.014,A -85,B 0,C 180,E1 -20161.762,E2 -20161.762} C_VEL
LIN {X 0,Y 228.283,Z 724.049,A -85,B 0,C 180,E1 -20167.074,E2 -20167.074} C_VEL
LIN {X 0,Y 228.097,Z 724.067,A -85,B 0,C 180,E1 -20170.653,E2 -20170.653} C_VEL
LIN {X 0,Y 227.991,Z 724.083,A -85,B 0,C 180,E1 -20176.107,E2 -20176.107} C_VEL
LIN {X 0,Y 227.874,Z 724.089,A -85,B 0,C 180,E1 -20179.363,E2 -20179.363} C_VEL
LIN {X 0,Y 227.228,Z 724.171,A -85,B 0,C 180,E1 -20180.839,E2 -20180.839} C_VEL
LIN {X 0,Y 224.429,Z 724.528,A -85,B 0,C 180,E1 -20183.249,E2 -20183.249} C_VEL
LIN {X 0,Y 221.177,Z 724.926,A -85,B 0,C 180,E1 -20186.225,E2 -20186.225} C_VEL
LIN {X 0,Y 220.811,Z 724.97,A -85,B 0,C 180,E1 -20187.255,E2 -20187.255} C_VEL
LIN {X 0,Y 220.788,Z 724.972,A -85,B 0,C 180,E1 -20190.776,E2 -20190.776} C_VEL
LIN {X 0,Y 220.767,Z 724.979,A -85,B 0,C 180,E1 -20194.961,E2 -20194.961} C_VEL
LIN {X 0,Y 220.837,Z 724.955,A -85,B 0,C 180,E1 -20199.797,E2 -20199.797} C_VEL
LIN {X 0,Y 220.866,Z 725.223,A -85,B 0,C 180,E1 -20200.057,E2 -20200.057} C_VEL
LIN {X 0,Y 223.324,Z 733.492,A -85,B 0,C 180,E1 -20203.816,E2 -20203.816} C_VEL
LIN {X 0,Y 225.891,Z 742.814,A -85,B 0,C 180,E1 -20207.687,E2 -20207.687} C_VEL
LIN {X 0,Y 227.958,Z 751.709,A -85,B 0,C 180,E1 -20211.091,E2 -20211.091} C_VEL
LIN {X 0,Y 229.238,Z 757.699,A -85,B 0,C 180,E1 -20213.221,E2 -20213.221} C_VEL
LIN {X 0,Y 233.806,Z 768.978,A -85,B 0,C 180,E1 -20214.437,E2 -20214.437} C_VEL
LIN {X 0,Y 237.152,Z 796.508,A -85,B 0,C 180,E1 -20215.972,E2 -20215.972} C_VEL
LIN {X 0,Y 239.88,Z 828.844,A -85,B 0,C 180,E1 -20217.514,E2 -20217.514} C_VEL
LIN {X 0,Y 240.534,Z 840.617,A -85,B 0,C 180,E1 -20218.012,E2 -20218.012} C_VEL
LIN {X 0,Y 239.291,Z 870.428,A -85,B 0,C 180,E1 -20218.914,E2 -20218.914} C_VEL
LIN {X 0,Y 237.879,Z 884.459,A -85,B 0,C 180,E1 -20219.653,E2 -20219.653} C_VEL
LIN {X 0,Y 236.177,Z 896.527,A -85,B 0,C 180,E1 -20220.609,E2 -20220.609} C_VEL
LIN {X 0,Y 233.695,Z 909.266,A -85,B 0,C 180,E1 -20221.987,E2 -20221.987} C_VEL
LIN {X 0,Y 231.091,Z 920.615,A -85,B 0,C 180,E1 -20223.606,E2 -20223.606} C_VEL
LIN {X 0,Y 228.454,Z 930.874,A -85,B 0,C 180,E1 -20225.476,E2 -20225.476} C_VEL
LIN {X 0,Y 225.888,Z 940.149,A -85,B 0,C 180,E1 -20227.611,E2 -20227.611} C_VEL
LIN {X 0,Y 223.871,Z 947.87,A -85,B 0,C 180,E1 -20229.813,E2 -20229.813} C_VEL
LIN {X 0,Y 221.922,Z 955.487,A -85,B 0,C 180,E1 -20232.505,E2 -20232.505} C_VEL
LIN {X 0,Y 220.657,Z 961.67,A -85,B 0,C 180,E1 -20235.252,E2 -20235.252} C_VEL
LIN {X 0,Y 219.893,Z 966.603,A -85,B 0,C 180,E1 -20238.023,E2 -20238.023} C_VEL
LIN {X 0,Y 219.644,Z 970.431,A -85,B 0,C 180,E1 -20240.807,E2 -20240.807} C_VEL
LIN {X 0,Y 219.776,Z 972.44,A -85,B 0,C 180,E1 -20242.664,E2 -20242.664} C_VEL
LIN {X 0,Y 219.992,Z 973.964,A -85,B 0,C 180,E1 -20244.513,E2 -20244.513} C_VEL
LIN {X 0,Y 220.271,Z 975.067,A -85,B 0,C 180,E1 -20246.354,E2 -20246.354} C_VEL
LIN {X 0,Y 220.488,Z 975.744,A -85,B 0,C 180,E1 -20248.186,E2 -20248.186} C_VEL
LIN {X 0,Y 220.733,Z 976.001,A -85,B 0,C 180,E1 -20250.012,E2 -20250.012} C_VEL
LIN {X 0,Y 220.484,Z 975.726,A -85,B 0,C 180,E1 -20251.839,E2 -20251.839} C_VEL
LIN {X 0,Y 220.262,Z 975.036,A -85,B 0,C 180,E1 -20253.671,E2 -20253.671} C_VEL
LIN {X 0,Y 219.945,Z 973.914,A -85,B 0,C 180,E1 -20255.513,E2 -20255.513} C_VEL
LIN {X 0,Y 219.726,Z 972.278,A -85,B 0,C 180,E1 -20257.456,E2 -20257.456} C_VEL
LIN {X 0,Y 219.753,Z 968.79,A -85,B 0,C 180,E1 -20260.608,E2 -20260.608} C_VEL
LIN {X 0,Y 220.081,Z 967.429,A -85,B 0,C 180,E1 -20262.928,E2 -20262.928} C_VEL
LIN {X 0,Y 221.458,Z 964.073,A -85,B 0,C 180,E1 -20266.607,E2 -20266.607} C_VEL
LIN {X 0,Y 224.115,Z 959.171,A -85,B 0,C 180,E1 -20270.19,E2 -20270.19} C_VEL
LIN {X 0,Y 226.943,Z 954.493,A -85,B 0,C 180,E1 -20272.785,E2 -20272.785} C_VEL
LIN {X 0,Y 231.066,Z 947.758,A -85,B 0,C 180,E1 -20275.696,E2 -20275.696} C_VEL
LIN {X 0,Y 235.366,Z 940.78,A -85,B 0,C 180,E1 -20278.064,E2 -20278.064} C_VEL
LIN {X 0,Y 239.456,Z 934.061,A -85,B 0,C 180,E1 -20279.941,E2 -20279.941} C_VEL
LIN {X 0,Y 244.893,Z 924.553,A -85,B 0,C 180,E1 -20282.078,E2 -20282.078} C_VEL
LIN {X 0,Y 249.968,Z 915.226,A -85,B 0,C 180,E1 -20283.74,E2 -20283.74} C_VEL
LIN {X 0,Y 254.917,Z 905.441,A -85,B 0,C 180,E1 -20285.146,E2 -20285.146} C_VEL
LIN {X 0,Y 259.562,Z 895.352,A -85,B 0,C 180,E1 -20286.33,E2 -20286.33} C_VEL
LIN {X 0,Y 263.891,Z 884.911,A -85,B 0,C 180,E1 -20287.302,E2 -20287.302} C_VEL
LIN {X 0,Y 268.164,Z 873.378,A -85,B 0,C 180,E1 -20288.165,E2 -20288.165} C_VEL
LIN {X 0,Y 272.597,Z 858.751,A -85,B 0,C 180,E1 -20289.062,E2 -20289.062} C_VEL
LIN {X 0,Y 275.267,Z 847.304,A -85,B 0,C 180,E1 -20289.674,E2 -20289.674} C_VEL
LIN {X 0,Y 277.901,Z 831.662,A -85,B 0,C 180,E1 -20290.837,E2 -20290.837} C_VEL
LIN {X 0,Y 280.365,Z 816.67,A -85,B 0,C 180,E1 -20292.295,E2 -20292.295} C_VEL
LIN {X 0,Y 282.672,Z 803.867,A -85,B 0,C 180,E1 -20293.744,E2 -20293.744} C_VEL
LIN {X 0,Y 283.178,Z 799.847,A -85,B 0,C 180,E1 -20294.889,E2 -20294.889} C_VEL
LIN {X 0,Y 283.043,Z 799.309,A -85,B 0,C 180,E1 -20296.07,E2 -20296.07} C_VEL
LIN {X 0,Y 283.342,Z 799.131,A -85,B 0,C 180,E1 -20298.093,E2 -20298.093} C_VEL
LIN {X 0,Y 284.361,Z 799.765,A -85,B 0,C 180,E1 -20300.159,E2 -20300.159} C_VEL
LIN {X 0,Y 284.521,Z 800.392,A -85,B 0,C 180,E1 -20300.55,E2 -20300.55} C_VEL
LIN {X 0,Y 279.705,Z 823.494,A -85,B 0,C 180,E1 -20301.827,E2 -20301.827} C_VEL
LIN {X 0,Y 276.951,Z 836.68,A -85,B 0,C 180,E1 -20302.738,E2 -20302.738} C_VEL
LIN {X 0,Y 273.717,Z 848.965,A -85,B 0,C 180,E1 -20303.804,E2 -20303.804} C_VEL
LIN {X 0,Y 269.91,Z 860.206,A -85,B 0,C 180,E1 -20305.051,E2 -20305.051} C_VEL
LIN {X 0,Y 265.74,Z 870.58,A -85,B 0,C 180,E1 -20306.49,E2 -20306.49} C_VEL
LIN {X 0,Y 261.673,Z 879.295,A -85,B 0,C 180,E1 -20307.964,E2 -20307.964} C_VEL
LIN {X 0,Y 256.528,Z 888.967,A -85,B 0,C 180,E1 -20310.001,E2 -20310.001} C_VEL
LIN {X 0,Y 251.577,Z 896.661,A -85,B 0,C 180,E1 -20312.1,E2 -20312.1} C_VEL
LIN {X 0,Y 247.747,Z 902.045,A -85,B 0,C 180,E1 -20313.915,E2 -20313.915} C_VEL
LIN {X 0,Y 243.42,Z 907.237,A -85,B 0,C 180,E1 -20316.159,E2 -20316.159} C_VEL
LIN {X 0,Y 239.441,Z 911.358,A -85,B 0,C 180,E1 -20318.476,E2 -20318.476} C_VEL
LIN {X 0,Y 235.79,Z 914.389,A -85,B 0,C 180,E1 -20320.861,E2 -20320.861} C_VEL
LIN {X 0,Y 233.572,Z 915.969,A -85,B 0,C 180,E1 -20322.489,E2 -20322.489} C_VEL
LIN {X 0,Y 229.64,Z 917.575,A -85,B 0,C 180,E1 -20325.828,E2 -20325.828} C_VEL
LIN {X 0,Y 227.928,Z 917.885,A -85,B 0,C 180,E1 -20327.535,E2 -20327.535} C_VEL
LIN {X 0,Y 226.389,Z 917.687,A -85,B 0,C 180,E1 -20329.265,E2 -20329.265} C_VEL
LIN {X 0,Y 224.072,Z 916.028,A -85,B 0,C 180,E1 -20332.793,E2 -20332.793} C_VEL
LIN {X 0,Y 223.247,Z 914.482,A -85,B 0,C 180,E1 -20334.581,E2 -20334.581} C_VEL
LIN {X 0,Y 222.069,Z 911.51,A -85,B 0,C 180,E1 -20337.279,E2 -20337.279} C_VEL
LIN {X 0,Y 221.496,Z 908.984,A -85,B 0,C 180,E1 -20339.091,E2 -20339.091} C_VEL
LIN {X 0,Y 220.927,Z 904.239,A -85,B 0,C 180,E1 -20341.823,E2 -20341.823} C_VEL
LIN {X 0,Y 220.684,Z 899.413,A -85,B 0,C 180,E1 -20344.109,E2 -20344.109} C_VEL
LIN {X 0,Y 220.877,Z 893.642,A -85,B 0,C 180,E1 -20346.394,E2 -20346.394} C_VEL
LIN {X 0,Y 221.331,Z 886.782,A -85,B 0,C 180,E1 -20348.675,E2 -20348.675} C_VEL
LIN {X 0,Y 221.751,Z 878.606,A -85,B 0,C 180,E1 -20350.962,E2 -20350.962} C_VEL
LIN {X 0,Y 222.35,Z 869.919,A -85,B 0,C 180,E1 -20353.015,E2 -20353.015} C_VEL
LIN {X 0,Y 223.007,Z 860.838,A -85,B 0,C 180,E1 -20354.836,E2 -20354.836} C_VEL
LIN {X 0,Y 223.607,Z 851.462,A -85,B 0,C 180,E1 -20356.432,E2 -20356.432} C_VEL
LIN {X 0,Y 224.33,Z 841.996,A -85,B 0,C 180,E1 -20357.786,E2 -20357.786} C_VEL
LIN {X 0,Y 224.974,Z 831.467,A -85,B 0,C 180,E1 -20359.03,E2 -20359.03} C_VEL
LIN {X 0,Y 225.489,Z 820.821,A -85,B 0,C 180,E1 -20360.051,E2 -20360.051} C_VEL
LIN {X 0,Y 225.963,Z 809.136,A -85,B 0,C 180,E1 -20360.921,E2 -20360.921} C_VEL
LIN {X 0,Y 226.556,Z 783.873,A -85,B 0,C 180,E1 -20362.274,E2 -20362.274} C_VEL
LIN {X 0,Y 227.791,Z 749.129,A -85,B 0,C 180,E1 -20364.037,E2 -20364.037} C_VEL
LIN {X 0,Y 220.947,Z 724.962,A -85,B 0,C 180,E1 -20365.641,E2 -20365.641} C_VEL
LIN {X 0,Y 220.848,Z 724.973,A -85,B 0,C 180,E1 -20370.754,E2 -20370.754} C_VEL
LIN {X 0,Y 220.82,Z 724.979,A -85,B 0,C 180,E1 -20374.952,E2 -20374.952} C_VEL
LIN {X 0,Y 220.829,Z 724.976,A -85,B 0,C 180,E1 -20377.27,E2 -20377.27} C_VEL
LIN {X 0,Y 220.773,Z 724.978,A -85,B 0,C 180,E1 -20381.952,E2 -20381.952} C_VEL
LIN {X 0,Y 220.777,Z 724.978,A -85,B 0,C 180,E1 -20385.534,E2 -20385.534} C_VEL
LIN {X 0,Y 220.805,Z 724.973,A -85,B 0,C 180,E1 -20390.45,E2 -20390.45} C_VEL
LIN {X 0,Y 220.848,Z 725.124,A -85,B 0,C 180,E1 -20392.437,E2 -20392.437} C_VEL
LIN {X 0,Y 221.897,Z 727.926,A -85,B 0,C 180,E1 -20392.766,E2 -20392.766} C_VEL
LIN {X 0,Y 223.641,Z 730.311,A -85,B 0,C 180,E1 -20393.212,E2 -20393.212} C_VEL
LIN {X 0,Y 230.438,Z 741.63,A -85,B 0,C 180,E1 -20394.941,E2 -20394.941} C_VEL
LIN {X 0,Y 237.377,Z 754.299,A -85,B 0,C 180,E1 -20396.609,E2 -20396.609} C_VEL
LIN {X 0,Y 243.134,Z 766.208,A -85,B 0,C 180,E1 -20397.946,E2 -20397.946} C_VEL
LIN {X 0,Y 242.213,Z 798.077,A -85,B 0,C 180,E1 -20398.904,E2 -20398.904} C_VEL
LIN {X 0,Y 241.828,Z 814.127,A -85,B 0,C 180,E1 -20399.51,E2 -20399.51} C_VEL
LIN {X 0,Y 241.118,Z 826.447,A -85,B 0,C 180,E1 -20400.286,E2 -20400.286} C_VEL
LIN {X 0,Y 239.676,Z 839.463,A -85,B 0,C 180,E1 -20401.45,E2 -20401.45} C_VEL
LIN {X 0,Y 237.975,Z 850.964,A -85,B 0,C 180,E1 -20402.827,E2 -20402.827} C_VEL
LIN {X 0,Y 235.92,Z 861.388,A -85,B 0,C 180,E1 -20404.398,E2 -20404.398} C_VEL
LIN {X 0,Y 234.038,Z 870.211,A -85,B 0,C 180,E1 -20406.073,E2 -20406.073} C_VEL
LIN {X 0,Y 231.89,Z 879.242,A -85,B 0,C 180,E1 -20408.195,E2 -20408.195} C_VEL
LIN {X 0,Y 229.389,Z 888.021,A -85,B 0,C 180,E1 -20410.759,E2 -20410.759} C_VEL
LIN {X 0,Y 227.076,Z 895.686,A -85,B 0,C 180,E1 -20413.628,E2 -20413.628} C_VEL
LIN {X 0,Y 225.446,Z 901.447,A -85,B 0,C 180,E1 -20416.468,E2 -20416.468} C_VEL
LIN {X 0,Y 224.543,Z 904.381,A -85,B 0,C 180,E1 -20418.25,E2 -20418.25} C_VEL
LIN {X 0,Y 223.087,Z 907.938,A -85,B 0,C 180,E1 -20420.926,E2 -20420.926} C_VEL
LIN {X 0,Y 222.44,Z 909.76,A -85,B 0,C 180,E1 -20422.728,E2 -20422.728} C_VEL
LIN {X 0,Y 221.873,Z 912.066,A -85,B 0,C 180,E1 -20426.356,E2 -20426.356} C_VEL
LIN {X 0,Y 221.529,Z 912.903,A -85,B 0,C 180,E1 -20429.988,E2 -20429.988} C_VEL
LIN {X 0,Y 221.867,Z 912.136,A -85,B 0,C 180,E1 -20433.62,E2 -20433.62} C_VEL
LIN {X 0,Y 222.416,Z 909.903,A -85,B 0,C 180,E1 -20437.249,E2 -20437.249} C_VEL
LIN {X 0,Y 223.488,Z 907.081,A -85,B 0,C 180,E1 -20439.947,E2 -20439.947} C_VEL
LIN {X 0,Y 224.908,Z 903.25,A -85,B 0,C 180,E1 -20442.622,E2 -20442.622} C_VEL
LIN {X 0,Y 226.536,Z 897.773,A -85,B 0,C 180,E1 -20445.563,E2 -20445.563} C_VEL
LIN {X 0,Y 228.616,Z 890.956,A -85,B 0,C 180,E1 -20448.353,E2 -20448.353} C_VEL
LIN {X 0,Y 230.983,Z 882.921,A -85,B 0,C 180,E1 -20450.934,E2 -20450.934} C_VEL
LIN {X 0,Y 233.092,Z 874.696,A -85,B 0,C 180,E1 -20453.063,E2 -20453.063} C_VEL
LIN {X 0,Y 235.378,Z 864.515,A -85,B 0,C 180,E1 -20455.167,E2 -20455.167} C_VEL
LIN {X 0,Y 237.532,Z 854.035,A -85,B 0,C 180,E1 -20456.868,E2 -20456.868} C_VEL
LIN {X 0,Y 239.482,Z 842.219,A -85,B 0,C 180,E1 -20458.376,E2 -20458.376} C_VEL
LIN {X 0,Y 240.986,Z 829.642,A -85,B 0,C 180,E1 -20459.574,E2 -20459.574} C_VEL
LIN {X 0,Y 241.808,Z 816.434,A -85,B 0,C 180,E1 -20460.5,E2 -20460.5} C_VEL
LIN {X 0,Y 242.201,Z 803.066,A -85,B 0,C 180,E1 -20461.069,E2 -20461.069} C_VEL
LIN {X 0,Y 243.145,Z 766.1,A -85,B 0,C 180,E1 -20462.198,E2 -20462.198} C_VEL
LIN {X 0,Y 235.881,Z 751.329,A -85,B 0,C 180,E1 -20463.895,E2 -20463.895} C_VEL
LIN {X 0,Y 227.155,Z 736.089,A -85,B 0,C 180,E1 -20466.033,E2 -20466.033} C_VEL
LIN {X 0,Y 222.729,Z 729.003,A -85,B 0,C 180,E1 -20467.18,E2 -20467.18} C_VEL
LIN {X 0,Y 221.119,Z 726.375,A -85,B 0,C 180,E1 -20467.615,E2 -20467.615} C_VEL
LIN {X 0,Y 220.796,Z 724.961,A -85,B 0,C 180,E1 -20467.777,E2 -20467.777} C_VEL
LIN {X 0,Y 220.837,Z 724.982,A -85,B 0,C 180,E1 -20471.917,E2 -20471.917} C_VEL
LIN {X 0,Y 220.834,Z 724.947,A -85,B 0,C 180,E1 -20475.561,E2 -20475.561} C_VEL
LIN {X 0,Y 220.817,Z 724.979,A -85,B 0,C 180,E1 -20479.782,E2 -20479.782} C_VEL
LIN {X 0,Y 220.788,Z 724.983,A -85,B 0,C 180,E1 -20482.786,E2 -20482.786} C_VEL
LIN {X 0,Y 220.773,Z 724.98,A -85,B 0,C 180,E1 -20487.236,E2 -20487.236} C_VEL
LIN {X 0,Y 220.774,Z 724.971,A -85,B 0,C 180,E1 -20491.477,E2 -20491.477} C_VEL
LIN {X 0,Y 220.807,Z 724.97,A -85,B 0,C 180,E1 -20495.558,E2 -20495.558} C_VEL
LIN {X 0,Y 220.826,Z 724.977,A -85,B 0,C 180,E1 -20499.507,E2 -20499.507} C_VEL
LIN {X 0,Y 220.954,Z 724.946,A -85,B 0,C 180,E1 -20503.365,E2 -20503.365} C_VEL
LIN {X 0,Y 221.028,Z 724.936,A -85,B 0,C 180,E1 -20509.001,E2 -20509.001} C_VEL
LIN {X 0,Y 221.216,Z 724.935,A -85,B 0,C 180,E1 -20512.699,E2 -20512.699} C_VEL
LIN {X 0,Y 221.459,Z 724.9,A -85,B 0,C 180,E1 -20518.181,E2 -20518.181} C_VEL
LIN {X 0,Y 221.459,Z 724.89,A -85,B 0,C 180,E1 -20521.818,E2 -20521.818} C_VEL
LIN {X 0,Y 221.216,Z 724.927,A -85,B 0,C 180,E1 -20527.301,E2 -20527.301} C_VEL
LIN {X 0,Y 221.045,Z 724.947,A -85,B 0,C 180,E1 -20530.997,E2 -20530.997} C_VEL
LIN {X 0,Y 220.954,Z 724.959,A -85,B 0,C 180,E1 -20536.635,E2 -20536.635} C_VEL
LIN {X 0,Y 220.833,Z 724.961,A -85,B 0,C 180,E1 -20540.492,E2 -20540.492} C_VEL
LIN {X 0,Y 220.811,Z 724.976,A -85,B 0,C 180,E1 -20544.442,E2 -20544.442} C_VEL
LIN {X 0,Y 220.811,Z 724.97,A -85,B 0,C 180,E1 -20547.255,E2 -20547.255} C_VEL
LIN {X 0,Y 220.079,Z 725.069,A -85,B 0,C 180,E1 -20548.776,E2 -20548.776} C_VEL
LIN {X 0,Y 217.226,Z 725.418,A -85,B 0,C 180,E1 -20551.26,E2 -20551.26} C_VEL
LIN {X 0,Y 214.029,Z 725.818,A -85,B 0,C 180,E1 -20554.33,E2 -20554.33} C_VEL
LIN {X 0,Y 213.704,Z 725.858,A -85,B 0,C 180,E1 -20555.393,E2 -20555.393} C_VEL
LIN {X 0,Y 213.734,Z 725.925,A -85,B 0,C 180,E1 -20558.664,E2 -20558.664} C_VEL
LIN {X 0,Y 216.496,Z 734.904,A -85,B 0,C 180,E1 -20562.978,E2 -20562.978} C_VEL
LIN {X 0,Y 218.929,Z 743.953,A -85,B 0,C 180,E1 -20566.913,E2 -20566.913} C_VEL
LIN {X 0,Y 220.701,Z 751.218,A -85,B 0,C 180,E1 -20569.841,E2 -20569.841} C_VEL
LIN {X 0,Y 221.868,Z 756.501,A -85,B 0,C 180,E1 -20571.788,E2 -20571.788} C_VEL
LIN {X 0,Y 228.081,Z 771.055,A -85,B 0,C 180,E1 -20573.518,E2 -20573.518} C_VEL
LIN {X 0,Y 231.282,Z 797.966,A -85,B 0,C 180,E1 -20575.074,E2 -20575.074} C_VEL
LIN {X 0,Y 233.964,Z 831.424,A -85,B 0,C 180,E1 -20576.713,E2 -20576.713} C_VEL
LIN {X 0,Y 234.423,Z 841.65,A -85,B 0,C 180,E1 -20577.146,E2 -20577.146} C_VEL
LIN {X 0,Y 233.201,Z 869.729,A -85,B 0,C 180,E1 -20578.024,E2 -20578.024} C_VEL
LIN {X 0,Y 231.745,Z 883.583,A -85,B 0,C 180,E1 -20578.772,E2 -20578.772} C_VEL
LIN {X 0,Y 229.999,Z 895.518,A -85,B 0,C 180,E1 -20579.739,E2 -20579.739} C_VEL
LIN {X 0,Y 227.777,Z 906.66,A -85,B 0,C 180,E1 -20580.94,E2 -20580.94} C_VEL
LIN {X 0,Y 225.015,Z 918.293,A -85,B 0,C 180,E1 -20582.584,E2 -20582.584} C_VEL
LIN {X 0,Y 222.226,Z 928.802,A -85,B 0,C 180,E1 -20584.491,E2 -20584.491} C_VEL
LIN {X 0,Y 219.778,Z 937.431,A -85,B 0,C 180,E1 -20586.454,E2 -20586.454} C_VEL
LIN {X 0,Y 217.531,Z 945.439,A -85,B 0,C 180,E1 -20588.702,E2 -20588.702} C_VEL
LIN {X 0,Y 215.74,Z 952.127,A -85,B 0,C 180,E1 -20591.003,E2 -20591.003} C_VEL
LIN {X 0,Y 214.134,Z 958.757,A -85,B 0,C 180,E1 -20593.815,E2 -20593.815} C_VEL
LIN {X 0,Y 213.071,Z 964.071,A -85,B 0,C 180,E1 -20596.664,E2 -20596.664} C_VEL
LIN {X 0,Y 212.607,Z 968.261,A -85,B 0,C 180,E1 -20599.538,E2 -20599.538} C_VEL
LIN {X 0,Y 212.7,Z 971.423,A -85,B 0,C 180,E1 -20602.418,E2 -20602.418} C_VEL
LIN {X 0,Y 212.897,Z 972.947,A -85,B 0,C 180,E1 -20604.329,E2 -20604.329} C_VEL
LIN {X 0,Y 213.213,Z 974.058,A -85,B 0,C 180,E1 -20606.233,E2 -20606.233} C_VEL
LIN {X 0,Y 213.435,Z 974.737,A -85,B 0,C 180,E1 -20608.126,E2 -20608.126} C_VEL
LIN {X 0,Y 213.694,Z 974.997,A -85,B 0,C 180,E1 -20610.012,E2 -20610.012} C_VEL
LIN {X 0,Y 213.43,Z 974.719,A -85,B 0,C 180,E1 -20611.899,E2 -20611.899} C_VEL
LIN {X 0,Y 213.199,Z 974.026,A -85,B 0,C 180,E1 -20613.792,E2 -20613.792} C_VEL
LIN {X 0,Y 212.678,Z 971.421,A -85,B 0,C 180,E1 -20617.537,E2 -20617.537} C_VEL
LIN {X 0,Y 212.772,Z 967.612,A -85,B 0,C 180,E1 -20620.96,E2 -20620.96} C_VEL
LIN {X 0,Y 213.13,Z 966.453,A -85,B 0,C 180,E1 -20623.358,E2 -20623.358} C_VEL
LIN {X 0,Y 214.606,Z 963.345,A -85,B 0,C 180,E1 -20627.153,E2 -20627.153} C_VEL
LIN {X 0,Y 216.123,Z 960.751,A -85,B 0,C 180,E1 -20629.432,E2 -20629.432} C_VEL
LIN {X 0,Y 218.402,Z 957.537,A -85,B 0,C 180,E1 -20631.731,E2 -20631.731} C_VEL
LIN {X 0,Y 221.52,Z 952.908,A -85,B 0,C 180,E1 -20634.37,E2 -20634.37} C_VEL
LIN {X 0,Y 226.045,Z 946.227,A -85,B 0,C 180,E1 -20637.308,E2 -20637.308} C_VEL
LIN {X 0,Y 230.832,Z 939.309,A -85,B 0,C 180,E1 -20639.664,E2 -20639.664} C_VEL
LIN {X 0,Y 236.103,Z 931.23,A -85,B 0,C 180,E1 -20641.905,E2 -20641.905} C_VEL
LIN {X 0,Y 242.1,Z 921.569,A -85,B 0,C 180,E1 -20643.984,E2 -20643.984} C_VEL
LIN {X 0,Y 246.995,Z 913.185,A -85,B 0,C 180,E1 -20645.443,E2 -20645.443} C_VEL
LIN {X 0,Y 252.874,Z 902.216,A -85,B 0,C 180,E1 -20646.953,E2 -20646.953} C_VEL
LIN {X 0,Y 257.817,Z 892.022,A -85,B 0,C 180,E1 -20648.089,E2 -20648.089} C_VEL
LIN {X 0,Y 262.241,Z 881.862,A -85,B 0,C 180,E1 -20648.969,E2 -20648.969} C_VEL
LIN {X 0,Y 267.847,Z 867.074,A -85,B 0,C 180,E1 -20650.015,E2 -20650.015} C_VEL
LIN {X 0,Y 272.179,Z 852.06,A -85,B 0,C 180,E1 -20650.848,E2 -20650.848} C_VEL
LIN {X 0,Y 275.205,Z 837.826,A -85,B 0,C 180,E1 -20651.842,E2 -20651.842} C_VEL
LIN {X 0,Y 277.653,Z 824.559,A -85,B 0,C 180,E1 -20653.062,E2 -20653.062} C_VEL
LIN {X 0,Y 280.521,Z 810.295,A -85,B 0,C 180,E1 -20654.602,E2 -20654.602} C_VEL
LIN {X 0,Y 280.975,Z 808.245,A -85,B 0,C 180,E1 -20654.885,E2 -20654.885} C_VEL
LIN {X 0,Y 281.317,Z 806.438,A -85,B 0,C 180,E1 -20655.39,E2 -20655.39} C_VEL
LIN {X 0,Y 281.404,Z 806.001,A -85,B 0,C 180,E1 -20657.599,E2 -20657.599} C_VEL
LIN {X 0,Y 282.079,Z 806.301,A -85,B 0,C 180,E1 -20659.403,E2 -20659.403} C_VEL
LIN {X 0,Y 277.412,Z 827.56,A -85,B 0,C 180,E1 -20660.612,E2 -20660.612} C_VEL
LIN {X 0,Y 274.129,Z 841.511,A -85,B 0,C 180,E1 -20661.617,E2 -20661.617} C_VEL
LIN {X 0,Y 270.744,Z 852.635,A -85,B 0,C 180,E1 -20662.644,E2 -20662.644} C_VEL
LIN {X 0,Y 267.191,Z 862.166,A -85,B 0,C 180,E1 -20663.713,E2 -20663.713} C_VEL
LIN {X 0,Y 263.269,Z 871.358,A -85,B 0,C 180,E1 -20664.974,E2 -20664.974} C_VEL
LIN {X 0,Y 259.408,Z 879.155,A -85,B 0,C 180,E1 -20666.262,E2 -20666.262} C_VEL
LIN {X 0,Y 254.727,Z 887.515,A -85,B 0,C 180,E1 -20667.919,E2 -20667.919} C_VEL
LIN {X 0,Y 250.269,Z 894.456,A -85,B 0,C 180,E1 -20669.637,E2 -20669.637} C_VEL
LIN {X 0,Y 245.998,Z 900.396,A -85,B 0,C 180,E1 -20671.41,E2 -20671.41} C_VEL
LIN {X 0,Y 241.96,Z 905.305,A -85,B 0,C 180,E1 -20673.242,E2 -20673.242} C_VEL
LIN {X 0,Y 237.456,Z 910.148,A -85,B 0,C 180,E1 -20675.521,E2 -20675.521} C_VEL
LIN {X 0,Y 233.249,Z 913.867,A -85,B 0,C 180,E1 -20677.875,E2 -20677.875} C_VEL
LIN {X 0,Y 229.426,Z 916.604,A -85,B 0,C 180,E1 -20680.308,E2 -20680.308} C_VEL
LIN {X 0,Y 224.957,Z 918.792,A -85,B 0,C 180,E1 -20683.67,E2 -20683.67} C_VEL
LIN {X 0,Y 221.138,Z 919.274,A -85,B 0,C 180,E1 -20687.146,E2 -20687.146} C_VEL
LIN {X 0,Y 219.538,Z 918.903,A -85,B 0,C 180,E1 -20688.926,E2 -20688.926} C_VEL
LIN {X 0,Y 218.217,Z 918.111,A -85,B 0,C 180,E1 -20690.733,E2 -20690.733} C_VEL
LIN {X 0,Y 216.233,Z 915.208,A -85,B 0,C 180,E1 -20694.405,E2 -20694.405} C_VEL
LIN {X 0,Y 214.72,Z 910.67,A -85,B 0,C 180,E1 -20698.124,E2 -20698.124} C_VEL
LIN {X 0,Y 213.981,Z 905.998,A -85,B 0,C 180,E1 -20700.941,E2 -20700.941} C_VEL
LIN {X 0,Y 213.616,Z 900.13,A -85,B 0,C 180,E1 -20703.773,E2 -20703.773} C_VEL
LIN {X 0,Y 213.815,Z 892.953,A -85,B 0,C 180,E1 -20706.606,E2 -20706.606} C_VEL
LIN {X 0,Y 214.223,Z 887.369,A -85,B 0,C 180,E1 -20708.49,E2 -20708.49} C_VEL
LIN {X 0,Y 214.577,Z 879.825,A -85,B 0,C 180,E1 -20710.663,E2 -20710.663} C_VEL
LIN {X 0,Y 215.233,Z 870.265,A -85,B 0,C 180,E1 -20712.973,E2 -20712.973} C_VEL
LIN {X 0,Y 215.906,Z 861.033,A -85,B 0,C 180,E1 -20714.853,E2 -20714.853} C_VEL
LIN {X 0,Y 216.515,Z 851.474,A -85,B 0,C 180,E1 -20716.501,E2 -20716.501} C_VEL
LIN {X 0,Y 217.271,Z 841.841,A -85,B 0,C 180,E1 -20717.896,E2 -20717.896} C_VEL
LIN {X 0,Y 218.01,Z 830.13,A -85,B 0,C 180,E1 -20719.295,E2 -20719.295} C_VEL
LIN {X 0,Y 218.679,Z 815.514,A -85,B 0,C 180,E1 -20720.642,E2 -20720.642} C_VEL
LIN {X 0,Y 219.173,Z 799.174,A -85,B 0,C 180,E1 -20721.673,E2 -20721.673} C_VEL
LIN {X 0,Y 220.711,Z 750.118,A -85,B 0,C 180,E1 -20724.265,E2 -20724.265} C_VEL
LIN {X 0,Y 213.892,Z 725.841,A -85,B 0,C 180,E1 -20725.957,E2 -20725.957} C_VEL
LIN {X 0,Y 213.797,Z 725.852,A -85,B 0,C 180,E1 -20731.258,E2 -20731.258} C_VEL
LIN {X 0,Y 213.794,Z 725.853,A -85,B 0,C 180,E1 -20734.716,E2 -20734.716} C_VEL
LIN {X 0,Y 213.73,Z 725.857,A -85,B 0,C 180,E1 -20738.666,E2 -20738.666} C_VEL
LIN {X 0,Y 213.727,Z 725.854,A -85,B 0,C 180,E1 -20743.648,E2 -20743.648} C_VEL
LIN {X 0,Y 213.726,Z 725.853,A -85,B 0,C 180,E1 -20746.339,E2 -20746.339} C_VEL
LIN {X 0,Y 213.769,Z 725.911,A -85,B 0,C 180,E1 -20750.94,E2 -20750.94} C_VEL
LIN {X 0,Y 214.786,Z 728.737,A -85,B 0,C 180,E1 -20751.288,E2 -20751.288} C_VEL
LIN {X 0,Y 216.647,Z 731.239,A -85,B 0,C 180,E1 -20751.801,E2 -20751.801} C_VEL
LIN {X 0,Y 223.847,Z 742.852,A -85,B 0,C 180,E1 -20753.75,E2 -20753.75} C_VEL
LIN {X 0,Y 231.209,Z 756.17,A -85,B 0,C 180,E1 -20755.625,E2 -20755.625} C_VEL
LIN {X 0,Y 237.074,Z 768.263,A -85,B 0,C 180,E1 -20757.06,E2 -20757.06} C_VEL
LIN {X 0,Y 236.239,Z 800.598,A -85,B 0,C 180,E1 -20758.079,E2 -20758.079} C_VEL
LIN {X 0,Y 235.762,Z 815.728,A -85,B 0,C 180,E1 -20758.67,E2 -20758.67} C_VEL
LIN {X 0,Y 234.916,Z 828.769,A -85,B 0,C 180,E1 -20759.544,E2 -20759.544} C_VEL
LIN {X 0,Y 233.376,Z 841.55,A -85,B 0,C 180,E1 -20760.74,E2 -20760.74} C_VEL
LIN {X 0,Y 231.52,Z 853.109,A -85,B 0,C 180,E1 -20762.184,E2 -20762.184} C_VEL
LIN {X 0,Y 229.388,Z 863.562,A -85,B 0,C 180,E1 -20763.858,E2 -20763.858} C_VEL
LIN {X 0,Y 227.13,Z 873.15,A -85,B 0,C 180,E1 -20765.785,E2 -20765.785} C_VEL
LIN {X 0,Y 224.945,Z 881.838,A -85,B 0,C 180,E1 -20767.97,E2 -20767.97} C_VEL
LIN {X 0,Y 222.386,Z 890.334,A -85,B 0,C 180,E1 -20770.609,E2 -20770.609} C_VEL
LIN {X 0,Y 220.183,Z 897.091,A -85,B 0,C 180,E1 -20773.294,E2 -20773.294} C_VEL
LIN {X 0,Y 218.619,Z 902.451,A -85,B 0,C 180,E1 -20776.037,E2 -20776.037} C_VEL
LIN {X 0,Y 217.668,Z 905.385,A -85,B 0,C 180,E1 -20777.874,E2 -20777.874} C_VEL
LIN {X 0,Y 216.15,Z 908.942,A -85,B 0,C 180,E1 -20780.632,E2 -20780.632} C_VEL
LIN {X 0,Y 215.47,Z 910.764,A -85,B 0,C 180,E1 -20782.491,E2 -20782.491} C_VEL
LIN {X 0,Y 214.86,Z 913.069,A -85,B 0,C 180,E1 -20786.237,E2 -20786.237} C_VEL
LIN {X 0,Y 214.501,Z 913.906,A -85,B 0,C 180,E1 -20789.988,E2 -20789.988} C_VEL
LIN {X 0,Y 214.853,Z 913.138,A -85,B 0,C 180,E1 -20793.738,E2 -20793.738} C_VEL
LIN {X 0,Y 215.445,Z 910.905,A -85,B 0,C 180,E1 -20797.484,E2 -20797.484} C_VEL
LIN {X 0,Y 216.57,Z 908.082,A -85,B 0,C 180,E1 -20800.268,E2 -20800.268} C_VEL
LIN {X 0,Y 218.055,Z 904.252,A -85,B 0,C 180,E1 -20803.025,E2 -20803.025} C_VEL
LIN {X 0,Y 219.774,Z 898.774,A -85,B 0,C 180,E1 -20806.054,E2 -20806.054} C_VEL
LIN {X 0,Y 221.956,Z 891.956,A -85,B 0,C 180,E1 -20808.925,E2 -20808.925} C_VEL
LIN {X 0,Y 224.433,Z 883.921,A -85,B 0,C 180,E1 -20811.575,E2 -20811.575} C_VEL
LIN {X 0,Y 226.642,Z 875.696,A -85,B 0,C 180,E1 -20813.759,E2 -20813.759} C_VEL
LIN {X 0,Y 229.046,Z 865.512,A -85,B 0,C 180,E1 -20815.913,E2 -20815.913} C_VEL
LIN {X 0,Y 231.291,Z 855.032,A -85,B 0,C 180,E1 -20817.654,E2 -20817.654} C_VEL
LIN {X 0,Y 233.32,Z 843.216,A -85,B 0,C 180,E1 -20819.197,E2 -20819.197} C_VEL
LIN {X 0,Y 234.897,Z 830.636,A -85,B 0,C 180,E1 -20820.42,E2 -20820.42} C_VEL
LIN {X 0,Y 235.781,Z 817.284,A -85,B 0,C 180,E1 -20821.376,E2 -20821.376} C_VEL
LIN {X 0,Y 236.191,Z 803.963,A -85,B 0,C 180,E1 -20821.954,E2 -20821.954} C_VEL
LIN {X 0,Y 237.154,Z 768.177,A -85,B 0,C 180,E1 -20823.076,E2 -20823.076} C_VEL
LIN {X 0,Y 229.744,Z 753.317,A -85,B 0,C 180,E1 -20824.894,E2 -20824.894} C_VEL
LIN {X 0,Y 222.192,Z 740.122,A -85,B 0,C 180,E1 -20826.842,E2 -20826.842} C_VEL
LIN {X 0,Y 218.032,Z 733.533,A -85,B 0,C 180,E1 -20827.968,E2 -20827.968} C_VEL
LIN {X 0,Y 215.811,Z 730.019,A -85,B 0,C 180,E1 -20828.595,E2 -20828.595} C_VEL
LIN {X 0,Y 214.139,Z 727.41,A -85,B 0,C 180,E1 -20829.077,E2 -20829.077} C_VEL
LIN {X 0,Y 213.777,Z 725.836,A -85,B 0,C 180,E1 -20829.26,E2 -20829.26} C_VEL
LIN {X 0,Y 213.799,Z 725.831,A -85,B 0,C 180,E1 -20833.681,E2 -20833.681} C_VEL
LIN {X 0,Y 213.8,Z 725.828,A -85,B 0,C 180,E1 -20836.345,E2 -20836.345} C_VEL
LIN {X 0,Y 213.781,Z 725.86,A -85,B 0,C 180,E1 -20839.1,E2 -20839.1} C_VEL
LIN {X 0,Y 213.707,Z 725.867,A -85,B 0,C 180,E1 -20843.704,E2 -20843.704} C_VEL
LIN {X 0,Y 213.72,Z 725.864,A -85,B 0,C 180,E1 -20848.254,E2 -20848.254} C_VEL
LIN {X 0,Y 213.774,Z 725.851,A -85,B 0,C 180,E1 -20852.596,E2 -20852.596} C_VEL
LIN {X 0,Y 213.764,Z 725.844,A -85,B 0,C 180,E1 -20856.968,E2 -20856.968} C_VEL
LIN {X 0,Y 213.884,Z 725.825,A -85,B 0,C 180,E1 -20862.798,E2 -20862.798} C_VEL
LIN {X 0,Y 213.89,Z 725.842,A -85,B 0,C 180,E1 -20866.702,E2 -20866.702} C_VEL
LIN {X 0,Y 214.09,Z 725.806,A -85,B 0,C 180,E1 -20870.553,E2 -20870.553} C_VEL
LIN {X 0,Y 214.154,Z 725.813,A -85,B 0,C 180,E1 -20872.457,E2 -20872.457} C_VEL
LIN {X 0,Y 214.417,Z 725.777,A -85,B 0,C 180,E1 -20878.122,E2 -20878.122} C_VEL
LIN {X 0,Y 214.417,Z 725.766,A -85,B 0,C 180,E1 -20881.878,E2 -20881.878} C_VEL
LIN {X 0,Y 214.154,Z 725.806,A -85,B 0,C 180,E1 -20887.543,E2 -20887.543} C_VEL
LIN {X 0,Y 213.962,Z 725.832,A -85,B 0,C 180,E1 -20891.366,E2 -20891.366} C_VEL
LIN {X 0,Y 213.868,Z 725.847,A -85,B 0,C 180,E1 -20895.242,E2 -20895.242} C_VEL
LIN {X 0,Y 213.78,Z 725.85,A -85,B 0,C 180,E1 -20899.193,E2 -20899.193} C_VEL
LIN {X 0,Y 213.774,Z 725.855,A -85,B 0,C 180,E1 -20903.235,E2 -20903.235} C_VEL
LIN {X 0,Y 213.777,Z 725.851,A -85,B 0,C 180,E1 -20907.457,E2 -20907.457} C_VEL
LIN {X 0,Y 213.719,Z 725.859,A -85,B 0,C 180,E1 -20911.746,E2 -20911.746} C_VEL
LIN {X 0,Y 213.704,Z 725.858,A -85,B 0,C 180,E1 -20915.393,E2 -20915.393} C_VEL
LIN {X 0,Y 213.469,Z 726.213,A -85,B 0,C 180,E1 -20916.436,E2 -20916.436} C_VEL
LIN {X 0,Y 212.581,Z 727.79,A -85,B 0,C 180,E1 -20917.947,E2 -20917.947} C_VEL
LIN {X 0,Y 211.446,Z 730.225,A -85,B 0,C 180,E1 -20919.382,E2 -20919.382} C_VEL
LIN {X 0,Y 210.203,Z 734.3,A -85,B 0,C 180,E1 -20921.264,E2 -20921.264} C_VEL
LIN {X 0,Y 210.056,Z 737.512,A -85,B 0,C 180,E1 -20922.669,E2 -20922.669} C_VEL
LIN {X 0,Y 210.247,Z 738.551,A -85,B 0,C 180,E1 -20923.14,E2 -20923.14} C_VEL
LIN {X 0,Y 212.366,Z 746.567,A -85,B 0,C 180,E1 -20926.724,E2 -20926.724} C_VEL
LIN {X 0,Y 214.409,Z 755.047,A -85,B 0,C 180,E1 -20930.197,E2 -20930.197} C_VEL
LIN {X 0,Y 216.556,Z 759.815,A -85,B 0,C 180,E1 -20930.849,E2 -20930.849} C_VEL
LIN {X 0,Y 222.553,Z 773.96,A -85,B 0,C 180,E1 -20932.611,E2 -20932.611} C_VEL
LIN {X 0,Y 225.61,Z 801.348,A -85,B 0,C 180,E1 -20934.228,E2 -20934.228} C_VEL
LIN {X 0,Y 228.174,Z 834.903,A -85,B 0,C 180,E1 -20935.918,E2 -20935.918} C_VEL
LIN {X 0,Y 228.358,Z 843.472,A -85,B 0,C 180,E1 -20936.262,E2 -20936.262} C_VEL
LIN {X 0,Y 227.237,Z 868.141,A -85,B 0,C 180,E1 -20937.047,E2 -20937.047} C_VEL
LIN {X 0,Y 225.824,Z 881.753,A -85,B 0,C 180,E1 -20937.785,E2 -20937.785} C_VEL
LIN {X 0,Y 224.057,Z 893.396,A -85,B 0,C 180,E1 -20938.717,E2 -20938.717} C_VEL
LIN {X 0,Y 221.598,Z 905.652,A -85,B 0,C 180,E1 -20940.048,E2 -20940.048} C_VEL
LIN {X 0,Y 218.723,Z 917.282,A -85,B 0,C 180,E1 -20941.725,E2 -20941.725} C_VEL
LIN {X 0,Y 215.832,Z 927.791,A -85,B 0,C 180,E1 -20943.678,E2 -20943.678} C_VEL
LIN {X 0,Y 213.267,Z 936.418,A -85,B 0,C 180,E1 -20945.69,E2 -20945.69} C_VEL
LIN {X 0,Y 210.872,Z 944.419,A -85,B 0,C 180,E1 -20947.994,E2 -20947.994} C_VEL
LIN {X 0,Y 208.666,Z 952.126,A -85,B 0,C 180,E1 -20950.77,E2 -20950.77} C_VEL
LIN {X 0,Y 206.816,Z 959.626,A -85,B 0,C 180,E1 -20954.24,E2 -20954.24} C_VEL
LIN {X 0,Y 205.874,Z 964.558,A -85,B 0,C 180,E1 -20957.194,E2 -20957.194} C_VEL
LIN {X 0,Y 205.513,Z 968.388,A -85,B 0,C 180,E1 -20960.169,E2 -20960.169} C_VEL
LIN {X 0,Y 205.64,Z 970.571,A -85,B 0,C 180,E1 -20962.357,E2 -20962.357} C_VEL
LIN {X 0,Y 206.151,Z 973.049,A -85,B 0,C 180,E1 -20966.104,E2 -20966.104} C_VEL
LIN {X 0,Y 206.38,Z 973.731,A -85,B 0,C 180,E1 -20968.062,E2 -20968.062} C_VEL
LIN {X 0,Y 206.653,Z 973.992,A -85,B 0,C 180,E1 -20970.013,E2 -20970.013} C_VEL
LIN {X 0,Y 206.374,Z 973.711,A -85,B 0,C 180,E1 -20971.964,E2 -20971.964} C_VEL
LIN {X 0,Y 206.115,Z 973.012,A -85,B 0,C 180,E1 -20973.923,E2 -20973.923} C_VEL
LIN {X 0,Y 205.618,Z 970.568,A -85,B 0,C 180,E1 -20977.599,E2 -20977.599} C_VEL
LIN {X 0,Y 205.823,Z 966.294,A -85,B 0,C 180,E1 -20981.585,E2 -20981.585} C_VEL
LIN {X 0,Y 206.847,Z 964.204,A -85,B 0,C 180,E1 -20985.785,E2 -20985.785} C_VEL
LIN {X 0,Y 209.212,Z 960.609,A -85,B 0,C 180,E1 -20989.848,E2 -20989.848} C_VEL
LIN {X 0,Y 212.814,Z 955.967,A -85,B 0,C 180,E1 -20993.358,E2 -20993.358} C_VEL
LIN {X 0,Y 216.334,Z 951.407,A -85,B 0,C 180,E1 -20996.025,E2 -20996.025} C_VEL
LIN {X 0,Y 221.389,Z 944.805,A -85,B 0,C 180,E1 -20998.966,E2 -20998.966} C_VEL
LIN {X 0,Y 227.431,Z 936.741,A -85,B 0,C 180,E1 -21001.702,E2 -21001.702} C_VEL
LIN {X 0,Y 232.191,Z 930.065,A -85,B 0,C 180,E1 -21003.543,E2 -21003.543} C_VEL
LIN {X 0,Y 237.475,Z 922.327,A -85,B 0,C 180,E1 -21005.258,E2 -21005.258} C_VEL
LIN {X 0,Y 243.759,Z 912.391,A -85,B 0,C 180,E1 -21007.014,E2 -21007.014} C_VEL
LIN {X 0,Y 249.27,Z 902.865,A -85,B 0,C 180,E1 -21008.347,E2 -21008.347} C_VEL
LIN {X 0,Y 254.408,Z 893.164,A -85,B 0,C 180,E1 -21009.458,E2 -21009.458} C_VEL
LIN {X 0,Y 259.034,Z 883.553,A -85,B 0,C 180,E1 -21010.325,E2 -21010.325} C_VEL
LIN {X 0,Y 264.785,Z 869.602,A -85,B 0,C 180,E1 -21011.328,E2 -21011.328} C_VEL
LIN {X 0,Y 269.718,Z 855.205,A -85,B 0,C 180,E1 -21012.169,E2 -21012.169} C_VEL
LIN {X 0,Y 271.41,Z 848.739,A -85,B 0,C 180,E1 -21012.564,E2 -21012.564} C_VEL
LIN {X 0,Y 274.283,Z 836.263,A -85,B 0,C 180,E1 -21013.526,E2 -21013.526} C_VEL
LIN {X 0,Y 277.196,Z 822.689,A -85,B 0,C 180,E1 -21014.853,E2 -21014.853} C_VEL
LIN {X 0,Y 279.424,Z 813.228,A -85,B 0,C 180,E1 -21015.909,E2 -21015.909} C_VEL
LIN {X 0,Y 279.795,Z 812.892,A -85,B 0,C 180,E1 -21018.241,E2 -21018.241} C_VEL
LIN {X 0,Y 274.229,Z 836.315,A -85,B 0,C 180,E1 -21019.695,E2 -21019.695} C_VEL
LIN {X 0,Y 271.099,Z 847.419,A -85,B 0,C 180,E1 -21020.569,E2 -21020.569} C_VEL
LIN {X 0,Y 267.927,Z 856.541,A -85,B 0,C 180,E1 -21021.465,E2 -21021.465} C_VEL
LIN {X 0,Y 263.179,Z 868.024,A -85,B 0,C 180,E1 -21022.83,E2 -21022.83} C_VEL
LIN {X 0,Y 257.513,Z 879.268,A -85,B 0,C 180,E1 -21024.553,E2 -21024.553} C_VEL
LIN {X 0,Y 252.505,Z 887.77,A -85,B 0,C 180,E1 -21026.175,E2 -21026.175} C_VEL
LIN {X 0,Y 247.7,Z 894.864,A -85,B 0,C 180,E1 -21027.86,E2 -21027.86} C_VEL
LIN {X 0,Y 243.128,Z 900.896,A -85,B 0,C 180,E1 -21029.611,E2 -21029.611} C_VEL
LIN {X 0,Y 237.866,Z 906.882,A -85,B 0,C 180,E1 -21031.788,E2 -21031.788} C_VEL
LIN {X 0,Y 233.025,Z 911.65,A -85,B 0,C 180,E1 -21034.067,E2 -21034.067} C_VEL
LIN {X 0,Y 228.475,Z 915.368,A -85,B 0,C 180,E1 -21036.429,E2 -21036.429} C_VEL
LIN {X 0,Y 223.082,Z 918.805,A -85,B 0,C 180,E1 -21039.724,E2 -21039.724} C_VEL
LIN {X 0,Y 218.345,Z 920.477,A -85,B 0,C 180,E1 -21043.161,E2 -21043.161} C_VEL
LIN {X 0,Y 216.266,Z 920.753,A -85,B 0,C 180,E1 -21044.931,E2 -21044.931} C_VEL
LIN {X 0,Y 214.35,Z 920.628,A -85,B 0,C 180,E1 -21046.732,E2 -21046.732} C_VEL
LIN {X 0,Y 212.689,Z 920.04,A -85,B 0,C 180,E1 -21048.565,E2 -21048.565} C_VEL
LIN {X 0,Y 211.295,Z 919.044,A -85,B 0,C 180,E1 -21050.427,E2 -21050.427} C_VEL
LIN {X 0,Y 209.205,Z 915.827,A -85,B 0,C 180,E1 -21054.216,E2 -21054.216} C_VEL
LIN {X 0,Y 207.95,Z 912.289,A -85,B 0,C 180,E1 -21057.094,E2 -21057.094} C_VEL
LIN {X 0,Y 206.983,Z 907.701,A -85,B 0,C 180,E1 -21060,E2 -21060} C_VEL
LIN {X 0,Y 206.599,Z 901.95,A -85,B 0,C 180,E1 -21062.925,E2 -21062.925} C_VEL
LIN {X 0,Y 206.597,Z 894.842,A -85,B 0,C 180,E1 -21065.858,E2 -21065.858} C_VEL
LIN {X 0,Y 207.092,Z 887.799,A -85,B 0,C 180,E1 -21068.293,E2 -21068.293} C_VEL
LIN {X 0,Y 207.421,Z 880.708,A -85,B 0,C 180,E1 -21070.391,E2 -21070.391} C_VEL
LIN {X 0,Y 208.02,Z 871.592,A -85,B 0,C 180,E1 -21072.686,E2 -21072.686} C_VEL
LIN {X 0,Y 208.704,Z 862.454,A -85,B 0,C 180,E1 -21074.629,E2 -21074.629} C_VEL
LIN {X 0,Y 209.356,Z 852.956,A -85,B 0,C 180,E1 -21076.329,E2 -21076.329} C_VEL
LIN {X 0,Y 210.082,Z 843.373,A -85,B 0,C 180,E1 -21077.774,E2 -21077.774} C_VEL
LIN {X 0,Y 210.723,Z 832.78,A -85,B 0,C 180,E1 -21079.103,E2 -21079.103} C_VEL
LIN {X 0,Y 211.214,Z 823.407,A -85,B 0,C 180,E1 -21080.069,E2 -21080.069} C_VEL
LIN {X 0,Y 211.751,Z 811.6,A -85,B 0,C 180,E1 -21081.031,E2 -21081.031} C_VEL
LIN {X 0,Y 212.414,Z 786.981,A -85,B 0,C 180,E1 -21082.486,E2 -21082.486} C_VEL
LIN {X 0,Y 213.668,Z 751.181,A -85,B 0,C 180,E1 -21084.483,E2 -21084.483} C_VEL
LIN {X 0,Y 206.936,Z 727.213,A -85,B 0,C 180,E1 -21086.141,E2 -21086.141} C_VEL
LIN {X 0,Y 206.868,Z 726.716,A -85,B 0,C 180,E1 -21086.21,E2 -21086.21} C_VEL
LIN {X 0,Y 206.737,Z 726.732,A -85,B 0,C 180,E1 -21091.784,E2 -21091.784} C_VEL
LIN {X 0,Y 206.729,Z 726.732,A -85,B 0,C 180,E1 -21095.306,E2 -21095.306} C_VEL
LIN {X 0,Y 206.673,Z 726.737,A -85,B 0,C 180,E1 -21100.249,E2 -21100.249} C_VEL
LIN {X 0,Y 206.655,Z 726.734,A -85,B 0,C 180,E1 -21104.41,E2 -21104.41} C_VEL
LIN {X 0,Y 206.694,Z 726.729,A -85,B 0,C 180,E1 -21109.295,E2 -21109.295} C_VEL
LIN {X 0,Y 207.668,Z 729.52,A -85,B 0,C 180,E1 -21109.671,E2 -21109.671} C_VEL
LIN {X 0,Y 209.494,Z 731.69,A -85,B 0,C 180,E1 -21110.206,E2 -21110.206} C_VEL
LIN {X 0,Y 211.609,Z 735.127,A -85,B 0,C 180,E1 -21110.848,E2 -21110.848} C_VEL
LIN {X 0,Y 219.048,Z 747.062,A -85,B 0,C 180,E1 -21112.961,E2 -21112.961} C_VEL
LIN {X 0,Y 226.854,Z 761.487,A -85,B 0,C 180,E1 -21115.043,E2 -21115.043} C_VEL
LIN {X 0,Y 231.12,Z 770.397,A -85,B 0,C 180,E1 -21116.139,E2 -21116.139} C_VEL
LIN {X 0,Y 230.307,Z 801.573,A -85,B 0,C 180,E1 -21117.153,E2 -21117.153} C_VEL
LIN {X 0,Y 229.797,Z 816.734,A -85,B 0,C 180,E1 -21117.76,E2 -21117.76} C_VEL
LIN {X 0,Y 228.879,Z 829.781,A -85,B 0,C 180,E1 -21118.651,E2 -21118.651} C_VEL
LIN {X 0,Y 227.27,Z 842.559,A -85,B 0,C 180,E1 -21119.874,E2 -21119.874} C_VEL
LIN {X 0,Y 225.328,Z 854.117,A -85,B 0,C 180,E1 -21121.35,E2 -21121.35} C_VEL
LIN {X 0,Y 223.101,Z 864.569,A -85,B 0,C 180,E1 -21123.063,E2 -21123.063} C_VEL
LIN {X 0,Y 220.74,Z 874.156,A -85,B 0,C 180,E1 -21125.037,E2 -21125.037} C_VEL
LIN {X 0,Y 218.446,Z 882.843,A -85,B 0,C 180,E1 -21127.278,E2 -21127.278} C_VEL
LIN {X 0,Y 215.769,Z 891.339,A -85,B 0,C 180,E1 -21129.989,E2 -21129.989} C_VEL
LIN {X 0,Y 213.462,Z 898.095,A -85,B 0,C 180,E1 -21132.752,E2 -21132.752} C_VEL
LIN {X 0,Y 211.806,Z 903.455,A -85,B 0,C 180,E1 -21135.578,E2 -21135.578} C_VEL
LIN {X 0,Y 210.802,Z 906.389,A -85,B 0,C 180,E1 -21137.472,E2 -21137.472} C_VEL
LIN {X 0,Y 209.219,Z 909.945,A -85,B 0,C 180,E1 -21140.319,E2 -21140.319} C_VEL
LIN {X 0,Y 208.504,Z 911.767,A -85,B 0,C 180,E1 -21142.239,E2 -21142.239} C_VEL
LIN {X 0,Y 207.848,Z 914.072,A -85,B 0,C 180,E1 -21146.11,E2 -21146.11} C_VEL
LIN {X 0,Y 207.474,Z 914.909,A -85,B 0,C 180,E1 -21149.987,E2 -21149.987} C_VEL
LIN {X 0,Y 207.841,Z 914.14,A -85,B 0,C 180,E1 -21153.865,E2 -21153.865} C_VEL
LIN {X 0,Y 208.479,Z 911.907,A -85,B 0,C 180,E1 -21157.736,E2 -21157.736} C_VEL
LIN {X 0,Y 209.659,Z 909.084,A -85,B 0,C 180,E1 -21160.61,E2 -21160.61} C_VEL
LIN {X 0,Y 211.214,Z 905.253,A -85,B 0,C 180,E1 -21163.455,E2 -21163.455} C_VEL
LIN {X 0,Y 213.029,Z 899.775,A -85,B 0,C 180,E1 -21166.577,E2 -21166.577} C_VEL
LIN {X 0,Y 215.32,Z 892.957,A -85,B 0,C 180,E1 -21169.531,E2 -21169.531} C_VEL
LIN {X 0,Y 217.912,Z 884.922,A -85,B 0,C 180,E1 -21172.254,E2 -21172.254} C_VEL
LIN {X 0,Y 220.228,Z 876.695,A -85,B 0,C 180,E1 -21174.495,E2 -21174.495} C_VEL
LIN {X 0,Y 222.749,Z 866.51,A -85,B 0,C 180,E1 -21176.703,E2 -21176.703} C_VEL
LIN {X 0,Y 225.084,Z 856.031,A -85,B 0,C 180,E1 -21178.485,E2 -21178.485} C_VEL
LIN {X 0,Y 227.211,Z 844.212,A -85,B 0,C 180,E1 -21180.061,E2 -21180.061} C_VEL
LIN {X 0,Y 228.863,Z 831.63,A -85,B 0,C 180,E1 -21181.311,E2 -21181.311} C_VEL
LIN {X 0,Y 229.816,Z 818.171,A -85,B 0,C 180,E1 -21182.295,E2 -21182.295} C_VEL
LIN {X 0,Y 230.25,Z 805.023,A -85,B 0,C 180,E1 -21182.878,E2 -21182.878} C_VEL
LIN {X 0,Y 231.202,Z 770.331,A -85,B 0,C 180,E1 -21183.999,E2 -21183.999} C_VEL
LIN {X 0,Y 224.078,Z 756.079,A -85,B 0,C 180,E1 -21185.84,E2 -21185.84} C_VEL
LIN {X 0,Y 215.888,Z 741.863,A -85,B 0,C 180,E1 -21188.079,E2 -21188.079} C_VEL
LIN {X 0,Y 211.182,Z 734.607,A -85,B 0,C 180,E1 -21189.44,E2 -21189.44} C_VEL
LIN {X 0,Y 208.992,Z 731.076,A -85,B 0,C 180,E1 -21190.111,E2 -21190.111} C_VEL
LIN {X 0,Y 207.297,Z 728.727,A -85,B 0,C 180,E1 -21190.627,E2 -21190.627} C_VEL
LIN {X 0,Y 206.743,Z 726.734,A -85,B 0,C 180,E1 -21190.89,E2 -21190.89} C_VEL
LIN {X 0,Y 206.706,Z 726.706,A -85,B 0,C 180,E1 -21195.539,E2 -21195.539} C_VEL
LIN {X 0,Y 206.701,Z 726.738,A -85,B 0,C 180,E1 -21199.758,E2 -21199.758} C_VEL
LIN {X 0,Y 206.685,Z 726.734,A -85,B 0,C 180,E1 -21204.686,E2 -21204.686} C_VEL
LIN {X 0,Y 206.657,Z 726.738,A -85,B 0,C 180,E1 -21209.328,E2 -21209.328} C_VEL
LIN {X 0,Y 206.678,Z 726.74,A -85,B 0,C 180,E1 -21213.764,E2 -21213.764} C_VEL
LIN {X 0,Y 206.683,Z 726.733,A -85,B 0,C 180,E1 -21218.035,E2 -21218.035} C_VEL
LIN {X 0,Y 206.814,Z 726.706,A -85,B 0,C 180,E1 -21222.191,E2 -21222.191} C_VEL
LIN {X 0,Y 206.832,Z 726.724,A -85,B 0,C 180,E1 -21226.24,E2 -21226.24} C_VEL
LIN {X 0,Y 207.04,Z 726.681,A -85,B 0,C 180,E1 -21230.228,E2 -21230.228} C_VEL
LIN {X 0,Y 207.009,Z 726.697,A -85,B 0,C 180,E1 -21234.154,E2 -21234.154} C_VEL
LIN {X 0,Y 207.35,Z 726.656,A -85,B 0,C 180,E1 -21238.058,E2 -21238.058} C_VEL
LIN {X 0,Y 207.457,Z 726.648,A -85,B 0,C 180,E1 -21240,E2 -21240} C_VEL
LIN {X 0,Y 207.35,Z 726.646,A -85,B 0,C 180,E1 -21241.942,E2 -21241.942} C_VEL
LIN {X 0,Y 207.094,Z 726.682,A -85,B 0,C 180,E1 -21247.802,E2 -21247.802} C_VEL
LIN {X 0,Y 206.882,Z 726.718,A -85,B 0,C 180,E1 -21251.761,E2 -21251.761} C_VEL
LIN {X 0,Y 206.802,Z 726.724,A -85,B 0,C 180,E1 -21255.776,E2 -21255.776} C_VEL
LIN {X 0,Y 206.709,Z 726.724,A -85,B 0,C 180,E1 -21259.877,E2 -21259.877} C_VEL
LIN {X 0,Y 206.701,Z 726.734,A -85,B 0,C 180,E1 -21264.08,E2 -21264.08} C_VEL
LIN {X 0,Y 206.685,Z 726.738,A -85,B 0,C 180,E1 -21268.428,E2 -21268.428} C_VEL
LIN {X 0,Y 206.656,Z 726.74,A -85,B 0,C 180,E1 -21272.965,E2 -21272.965} C_VEL
